    movel(p[x_c + -0.041312, y_c + 0.071568, z_c, rx, ry, rz], a, v)
    movel(p[x_c + -0.041015, y_c + 0.071951, z_c, rx, ry, rz], a, v)
    movel(p[x_c + -0.040710, y_c + 0.072343, z_c, rx, ry, rz], a, v)
    movel(p[x_c + -0.040396, y_c + 0.072744, z_c, rx, ry, rz], a, v)
    movel(p[x_c + -0.040073, y_c + 0.073156, z_c, rx, ry, rz], a, v)
    movel(p[x_c + -0.040073, y_c + 0.073156, z_c, rx, ry, rz], a, v)
    movel(p[x_c + -0.039958, y_c + 0.073302, z_c, rx, ry, rz], a, v)
    movel(p[x_c + -0.039844, y_c + 0.073448, z_c, rx, ry, rz], a, v)
    movel(p[x_c + -0.039729, y_c + 0.073594, z_c, rx, ry, rz], a, v)
    movel(p[x_c + -0.039615, y_c + 0.073740, z_c, rx, ry, rz], a, v)
    movel(p[x_c + -0.039501, y_c + 0.073885, z_c, rx, ry, rz], a, v)
    movel(p[x_c + -0.039388, y_c + 0.074029, z_c, rx, ry, rz], a, v)
    movel(p[x_c + -0.039276, y_c + 0.074172, z_c, rx, ry, rz], a, v)
    movel(p[x_c + -0.039164, y_c + 0.074315, z_c, rx, ry, rz], a, v)
    movel(p[x_c + -0.039053, y_c + 0.074457, z_c, rx, ry, rz], a, v)
    movel(p[x_c + -0.038942, y_c + 0.074597, z_c, rx, ry, rz], a, v)
    movel(p[x_c + -0.038833, y_c + 0.074737, z_c, rx, ry, rz], a, v)
    movel(p[x_c + -0.038724, y_c + 0.074876, z_c, rx, ry, rz], a, v)
    movel(p[x_c + -0.038617, y_c + 0.075013, z_c, rx, ry, rz], a, v)
    movel(p[x_c + -0.038511, y_c + 0.075148, z_c, rx, ry, rz], a, v)
    movel(p[x_c + -0.038405, y_c + 0.075283, z_c, rx, ry, rz], a, v)
    movel(p[x_c + -0.038301, y_c + 0.075416, z_c, rx, ry, rz], a, v)
    movel(p[x_c + -0.038199, y_c + 0.075547, z_c, rx, ry, rz], a, v)
    movel(p[x_c + -0.038098, y_c + 0.075676, z_c, rx, ry, rz], a, v)
    movel(p[x_c + -0.037998, y_c + 0.075804, z_c, rx, ry, rz], a, v)
    movel(p[x_c + -0.037900, y_c + 0.075929, z_c, rx, ry, rz], a, v)
    movel(p[x_c + -0.037803, y_c + 0.076053, z_c, rx, ry, rz], a, v)
    movel(p[x_c + -0.037708, y_c + 0.076174, z_c, rx, ry, rz], a, v)
    movel(p[x_c + -0.037615, y_c + 0.076294, z_c, rx, ry, rz], a, v)
    movel(p[x_c + -0.037523, y_c + 0.076411, z_c, rx, ry, rz], a, v)
    movel(p[x_c + -0.037434, y_c + 0.076525, z_c, rx, ry, rz], a, v)
    movel(p[x_c + -0.037346, y_c + 0.076637, z_c, rx, ry, rz], a, v)
    movel(p[x_c + -0.037261, y_c + 0.076747, z_c, rx, ry, rz], a, v)
    movel(p[x_c + -0.037177, y_c + 0.076854, z_c, rx, ry, rz], a, v)
    movel(p[x_c + -0.037096, y_c + 0.076958, z_c, rx, ry, rz], a, v)
    movel(p[x_c + -0.037017, y_c + 0.077059, z_c, rx, ry, rz], a, v)
    movel(p[x_c + -0.036940, y_c + 0.077157, z_c, rx, ry, rz], a, v)
    movel(p[x_c + -0.036866, y_c + 0.077253, z_c, rx, ry, rz], a, v)
    movel(p[x_c + -0.036794, y_c + 0.077345, z_c, rx, ry, rz], a, v)
    movel(p[x_c + -0.036725, y_c + 0.077434, z_c, rx, ry, rz], a, v)
    movel(p[x_c + -0.036658, y_c + 0.077519, z_c, rx, ry, rz], a, v)
    movel(p[x_c + -0.036594, y_c + 0.077602, z_c, rx, ry, rz], a, v)
    movel(p[x_c + -0.036533, y_c + 0.077680, z_c, rx, ry, rz], a, v)
    movel(p[x_c + -0.036475, y_c + 0.077755, z_c, rx, ry, rz], a, v)
    movel(p[x_c + -0.036419, y_c + 0.077827, z_c, rx, ry, rz], a, v)
    movel(p[x_c + -0.036367, y_c + 0.077895, z_c, rx, ry, rz], a, v)
    movel(p[x_c + -0.036317, y_c + 0.077959, z_c, rx, ry, rz], a, v)
    movel(p[x_c + -0.036271, y_c + 0.078018, z_c, rx, ry, rz], a, v)
    movel(p[x_c + -0.036227, y_c + 0.078074, z_c, rx, ry, rz], a, v)
    movel(p[x_c + -0.036188, y_c + 0.078126, z_c, rx, ry, rz], a, v)
    movel(p[x_c + -0.036151, y_c + 0.078173, z_c, rx, ry, rz], a, v)
    movel(p[x_c + -0.036118, y_c + 0.078217, z_c, rx, ry, rz], a, v)
    movel(p[x_c + -0.036088, y_c + 0.078255, z_c, rx, ry, rz], a, v)
    movel(p[x_c + -0.036062, y_c + 0.078290, z_c, rx, ry, rz], a, v)
    movel(p[x_c + -0.036039, y_c + 0.078319, z_c, rx, ry, rz], a, v)
    movel(p[x_c + -0.036039, y_c + 0.078319, z_c, rx, ry, rz], a, v)
    movel(p[x_c + -0.035423, y_c + 0.079129, z_c, rx, ry, rz], a, v)
    movel(p[x_c + -0.035423, y_c + 0.079129, z_c, rx, ry, rz], a, v)
    movel(p[x_c + -0.037378, y_c + 0.080396, z_c, rx, ry, rz], a, v)
    movel(p[x_c + -0.037378, y_c + 0.080396, z_c, rx, ry, rz], a, v)
    movel(p[x_c + -0.037680, y_c + 0.080589, z_c, rx, ry, rz], a, v)
    movel(p[x_c + -0.037987, y_c + 0.080780, z_c, rx, ry, rz], a, v)
    movel(p[x_c + -0.038299, y_c + 0.080970, z_c, rx, ry, rz], a, v)
    movel(p[x_c + -0.038617, y_c + 0.081159, z_c, rx, ry, rz], a, v)
    movel(p[x_c + -0.038940, y_c + 0.081346, z_c, rx, ry, rz], a, v)
    movel(p[x_c + -0.039269, y_c + 0.081532, z_c, rx, ry, rz], a, v)
    movel(p[x_c + -0.039602, y_c + 0.081716, z_c, rx, ry, rz], a, v)
    movel(p[x_c + -0.039939, y_c + 0.081898, z_c, rx, ry, rz], a, v)
    movel(p[x_c + -0.040281, y_c + 0.082078, z_c, rx, ry, rz], a, v)
    movel(p[x_c + -0.040628, y_c + 0.082257, z_c, rx, ry, rz], a, v)
    movel(p[x_c + -0.040978, y_c + 0.082434, z_c, rx, ry, rz], a, v)
    movel(p[x_c + -0.041332, y_c + 0.082609, z_c, rx, ry, rz], a, v)
    movel(p[x_c + -0.041690, y_c + 0.082782, z_c, rx, ry, rz], a, v)
    movel(p[x_c + -0.042052, y_c + 0.082952, z_c, rx, ry, rz], a, v)
    movel(p[x_c + -0.042417, y_c + 0.083121, z_c, rx, ry, rz], a, v)
    movel(p[x_c + -0.042785, y_c + 0.083287, z_c, rx, ry, rz], a, v)
    movel(p[x_c + -0.043157, y_c + 0.083452, z_c, rx, ry, rz], a, v)
    movel(p[x_c + -0.043531, y_c + 0.083613, z_c, rx, ry, rz], a, v)
    movel(p[x_c + -0.043908, y_c + 0.083773, z_c, rx, ry, rz], a, v)
    movel(p[x_c + -0.044287, y_c + 0.083930, z_c, rx, ry, rz], a, v)
    movel(p[x_c + -0.044668, y_c + 0.084084, z_c, rx, ry, rz], a, v)
    movel(p[x_c + -0.045052, y_c + 0.084236, z_c, rx, ry, rz], a, v)
    movel(p[x_c + -0.045438, y_c + 0.084385, z_c, rx, ry, rz], a, v)
    movel(p[x_c + -0.045825, y_c + 0.084531, z_c, rx, ry, rz], a, v)
    movel(p[x_c + -0.046214, y_c + 0.084674, z_c, rx, ry, rz], a, v)
    movel(p[x_c + -0.046604, y_c + 0.084815, z_c, rx, ry, rz], a, v)
    movel(p[x_c + -0.046996, y_c + 0.084952, z_c, rx, ry, rz], a, v)
    movel(p[x_c + -0.047388, y_c + 0.085087, z_c, rx, ry, rz], a, v)
    movel(p[x_c + -0.047782, y_c + 0.085219, z_c, rx, ry, rz], a, v)
    movel(p[x_c + -0.048176, y_c + 0.085347, z_c, rx, ry, rz], a, v)
    movel(p[x_c + -0.048571, y_c + 0.085472, z_c, rx, ry, rz], a, v)
    movel(p[x_c + -0.048966, y_c + 0.085594, z_c, rx, ry, rz], a, v)
    movel(p[x_c + -0.049361, y_c + 0.085713, z_c, rx, ry, rz], a, v)
    movel(p[x_c + -0.049756, y_c + 0.085828, z_c, rx, ry, rz], a, v)
    movel(p[x_c + -0.050151, y_c + 0.085939, z_c, rx, ry, rz], a, v)
    movel(p[x_c + -0.050545, y_c + 0.086047, z_c, rx, ry, rz], a, v)
    movel(p[x_c + -0.050939, y_c + 0.086152, z_c, rx, ry, rz], a, v)
    movel(p[x_c + -0.051332, y_c + 0.086253, z_c, rx, ry, rz], a, v)
    movel(p[x_c + -0.051724, y_c + 0.086350, z_c, rx, ry, rz], a, v)
    movel(p[x_c + -0.052115, y_c + 0.086443, z_c, rx, ry, rz], a, v)
    movel(p[x_c + -0.052505, y_c + 0.086532, z_c, rx, ry, rz], a, v)
    movel(p[x_c + -0.052893, y_c + 0.086618, z_c, rx, ry, rz], a, v)
    movel(p[x_c + -0.053280, y_c + 0.086699, z_c, rx, ry, rz], a, v)
    movel(p[x_c + -0.053665, y_c + 0.086777, z_c, rx, ry, rz], a, v)
    movel(p[x_c + -0.054047, y_c + 0.086850, z_c, rx, ry, rz], a, v)
    movel(p[x_c + -0.054428, y_c + 0.086919, z_c, rx, ry, rz], a, v)
    movel(p[x_c + -0.054806, y_c + 0.086984, z_c, rx, ry, rz], a, v)
    movel(p[x_c + -0.055182, y_c + 0.087044, z_c, rx, ry, rz], a, v)
    movel(p[x_c + -0.055554, y_c + 0.087100, z_c, rx, ry, rz], a, v)
    movel(p[x_c + -0.055554, y_c + 0.087100, z_c, rx, ry, rz], a, v)
    movel(p[x_c + -0.055822, y_c + 0.087137, z_c, rx, ry, rz], a, v)
    movel(p[x_c + -0.056094, y_c + 0.087172, z_c, rx, ry, rz], a, v)
    movel(p[x_c + -0.056371, y_c + 0.087205, z_c, rx, ry, rz], a, v)
    movel(p[x_c + -0.056652, y_c + 0.087236, z_c, rx, ry, rz], a, v)
    movel(p[x_c + -0.056937, y_c + 0.087265, z_c, rx, ry, rz], a, v)
    movel(p[x_c + -0.057226, y_c + 0.087292, z_c, rx, ry, rz], a, v)
    movel(p[x_c + -0.057519, y_c + 0.087317, z_c, rx, ry, rz], a, v)
    movel(p[x_c + -0.057816, y_c + 0.087340, z_c, rx, ry, rz], a, v)
    movel(p[x_c + -0.058116, y_c + 0.087360, z_c, rx, ry, rz], a, v)
    movel(p[x_c + -0.058421, y_c + 0.087379, z_c, rx, ry, rz], a, v)
    movel(p[x_c + -0.058728, y_c + 0.087395, z_c, rx, ry, rz], a, v)
    movel(p[x_c + -0.059039, y_c + 0.087410, z_c, rx, ry, rz], a, v)
    movel(p[x_c + -0.059354, y_c + 0.087422, z_c, rx, ry, rz], a, v)
    movel(p[x_c + -0.059671, y_c + 0.087432, z_c, rx, ry, rz], a, v)
    movel(p[x_c + -0.059991, y_c + 0.087441, z_c, rx, ry, rz], a, v)
    movel(p[x_c + -0.060315, y_c + 0.087447, z_c, rx, ry, rz], a, v)
    movel(p[x_c + -0.060641, y_c + 0.087451, z_c, rx, ry, rz], a, v)
    movel(p[x_c + -0.060969, y_c + 0.087453, z_c, rx, ry, rz], a, v)
    movel(p[x_c + -0.061300, y_c + 0.087453, z_c, rx, ry, rz], a, v)
    movel(p[x_c + -0.061634, y_c + 0.087451, z_c, rx, ry, rz], a, v)
    movel(p[x_c + -0.061970, y_c + 0.087447, z_c, rx, ry, rz], a, v)
    movel(p[x_c + -0.062308, y_c + 0.087441, z_c, rx, ry, rz], a, v)
    movel(p[x_c + -0.062648, y_c + 0.087433, z_c, rx, ry, rz], a, v)
    movel(p[x_c + -0.062990, y_c + 0.087423, z_c, rx, ry, rz], a, v)
    movel(p[x_c + -0.063334, y_c + 0.087411, z_c, rx, ry, rz], a, v)
    movel(p[x_c + -0.063679, y_c + 0.087397, z_c, rx, ry, rz], a, v)
    movel(p[x_c + -0.064027, y_c + 0.087381, z_c, rx, ry, rz], a, v)
    movel(p[x_c + -0.064375, y_c + 0.087363, z_c, rx, ry, rz], a, v)
    movel(p[x_c + -0.064725, y_c + 0.087343, z_c, rx, ry, rz], a, v)
    movel(p[x_c + -0.065076, y_c + 0.087321, z_c, rx, ry, rz], a, v)
    movel(p[x_c + -0.065428, y_c + 0.087297, z_c, rx, ry, rz], a, v)
    movel(p[x_c + -0.065782, y_c + 0.087271, z_c, rx, ry, rz], a, v)
    movel(p[x_c + -0.066136, y_c + 0.087243, z_c, rx, ry, rz], a, v)
    movel(p[x_c + -0.066491, y_c + 0.087213, z_c, rx, ry, rz], a, v)
    movel(p[x_c + -0.066846, y_c + 0.087181, z_c, rx, ry, rz], a, v)
    movel(p[x_c + -0.067202, y_c + 0.087148, z_c, rx, ry, rz], a, v)
    movel(p[x_c + -0.067558, y_c + 0.087112, z_c, rx, ry, rz], a, v)
    movel(p[x_c + -0.067915, y_c + 0.087074, z_c, rx, ry, rz], a, v)
    movel(p[x_c + -0.068272, y_c + 0.087034, z_c, rx, ry, rz], a, v)
    movel(p[x_c + -0.068629, y_c + 0.086993, z_c, rx, ry, rz], a, v)
    movel(p[x_c + -0.068985, y_c + 0.086949, z_c, rx, ry, rz], a, v)
    movel(p[x_c + -0.069342, y_c + 0.086904, z_c, rx, ry, rz], a, v)
    movel(p[x_c + -0.069698, y_c + 0.086856, z_c, rx, ry, rz], a, v)
    movel(p[x_c + -0.070054, y_c + 0.086807, z_c, rx, ry, rz], a, v)
    movel(p[x_c + -0.070409, y_c + 0.086755, z_c, rx, ry, rz], a, v)
    movel(p[x_c + -0.070764, y_c + 0.086702, z_c, rx, ry, rz], a, v)
    movel(p[x_c + -0.071117, y_c + 0.086647, z_c, rx, ry, rz], a, v)
    movel(p[x_c + -0.071470, y_c + 0.086590, z_c, rx, ry, rz], a, v)
    movel(p[x_c + -0.071822, y_c + 0.086531, z_c, rx, ry, rz], a, v)
    movel(p[x_c + -0.071822, y_c + 0.086531, z_c, rx, ry, rz], a, v)
    movel(p[x_c + -0.071990, y_c + 0.086502, z_c, rx, ry, rz], a, v)
    movel(p[x_c + -0.072167, y_c + 0.086470, z_c, rx, ry, rz], a, v)
    movel(p[x_c + -0.072353, y_c + 0.086437, z_c, rx, ry, rz], a, v)
    movel(p[x_c + -0.072546, y_c + 0.086401, z_c, rx, ry, rz], a, v)
    movel(p[x_c + -0.072747, y_c + 0.086363, z_c, rx, ry, rz], a, v)
    movel(p[x_c + -0.072956, y_c + 0.086323, z_c, rx, ry, rz], a, v)
    movel(p[x_c + -0.073172, y_c + 0.086281, z_c, rx, ry, rz], a, v)
    movel(p[x_c + -0.073394, y_c + 0.086237, z_c, rx, ry, rz], a, v)
    movel(p[x_c + -0.073623, y_c + 0.086191, z_c, rx, ry, rz], a, v)
    movel(p[x_c + -0.073857, y_c + 0.086144, z_c, rx, ry, rz], a, v)
    movel(p[x_c + -0.074097, y_c + 0.086095, z_c, rx, ry, rz], a, v)
    movel(p[x_c + -0.074342, y_c + 0.086045, z_c, rx, ry, rz], a, v)
    movel(p[x_c + -0.074591, y_c + 0.085993, z_c, rx, ry, rz], a, v)
    movel(p[x_c + -0.074845, y_c + 0.085940, z_c, rx, ry, rz], a, v)
    movel(p[x_c + -0.075103, y_c + 0.085885, z_c, rx, ry, rz], a, v)
    movel(p[x_c + -0.075365, y_c + 0.085830, z_c, rx, ry, rz], a, v)
    movel(p[x_c + -0.075629, y_c + 0.085773, z_c, rx, ry, rz], a, v)
    movel(p[x_c + -0.075897, y_c + 0.085716, z_c, rx, ry, rz], a, v)
    movel(p[x_c + -0.076166, y_c + 0.085657, z_c, rx, ry, rz], a, v)
    movel(p[x_c + -0.076438, y_c + 0.085598, z_c, rx, ry, rz], a, v)
    movel(p[x_c + -0.076712, y_c + 0.085538, z_c, rx, ry, rz], a, v)
    movel(p[x_c + -0.076986, y_c + 0.085477, z_c, rx, ry, rz], a, v)
    movel(p[x_c + -0.077262, y_c + 0.085416, z_c, rx, ry, rz], a, v)
    movel(p[x_c + -0.077538, y_c + 0.085354, z_c, rx, ry, rz], a, v)
    movel(p[x_c + -0.077814, y_c + 0.085292, z_c, rx, ry, rz], a, v)
    movel(p[x_c + -0.078090, y_c + 0.085229, z_c, rx, ry, rz], a, v)
    movel(p[x_c + -0.078365, y_c + 0.085167, z_c, rx, ry, rz], a, v)
    movel(p[x_c + -0.078640, y_c + 0.085104, z_c, rx, ry, rz], a, v)
    movel(p[x_c + -0.078912, y_c + 0.085041, z_c, rx, ry, rz], a, v)
    movel(p[x_c + -0.079184, y_c + 0.084978, z_c, rx, ry, rz], a, v)
    movel(p[x_c + -0.079452, y_c + 0.084916, z_c, rx, ry, rz], a, v)
    movel(p[x_c + -0.079719, y_c + 0.084853, z_c, rx, ry, rz], a, v)
    movel(p[x_c + -0.079982, y_c + 0.084791, z_c, rx, ry, rz], a, v)
    movel(p[x_c + -0.080242, y_c + 0.084729, z_c, rx, ry, rz], a, v)
    movel(p[x_c + -0.080499, y_c + 0.084668, z_c, rx, ry, rz], a, v)
    movel(p[x_c + -0.080751, y_c + 0.084607, z_c, rx, ry, rz], a, v)
    movel(p[x_c + -0.080999, y_c + 0.084547, z_c, rx, ry, rz], a, v)
    movel(p[x_c + -0.081242, y_c + 0.084488, z_c, rx, ry, rz], a, v)
    movel(p[x_c + -0.081480, y_c + 0.084429, z_c, rx, ry, rz], a, v)
    movel(p[x_c + -0.081712, y_c + 0.084372, z_c, rx, ry, rz], a, v)
    movel(p[x_c + -0.081938, y_c + 0.084315, z_c, rx, ry, rz], a, v)
    movel(p[x_c + -0.082158, y_c + 0.084259, z_c, rx, ry, rz], a, v)
    movel(p[x_c + -0.082371, y_c + 0.084205, z_c, rx, ry, rz], a, v)
    movel(p[x_c + -0.082577, y_c + 0.084152, z_c, rx, ry, rz], a, v)
    movel(p[x_c + -0.082775, y_c + 0.084100, z_c, rx, ry, rz], a, v)
    movel(p[x_c + -0.082965, y_c + 0.084049, z_c, rx, ry, rz], a, v)
    movel(p[x_c + -0.083148, y_c + 0.084000, z_c, rx, ry, rz], a, v)
    movel(p[x_c + -0.083321, y_c + 0.083953, z_c, rx, ry, rz], a, v)
    movel(p[x_c + -0.083486, y_c + 0.083907, z_c, rx, ry, rz], a, v)
    movel(p[x_c + -0.083486, y_c + 0.083907, z_c, rx, ry, rz], a, v)
    movel(p[x_c + -0.083592, y_c + 0.083878, z_c, rx, ry, rz], a, v)
    movel(p[x_c + -0.083694, y_c + 0.083849, z_c, rx, ry, rz], a, v)
    movel(p[x_c + -0.083792, y_c + 0.083822, z_c, rx, ry, rz], a, v)
    movel(p[x_c + -0.083885, y_c + 0.083797, z_c, rx, ry, rz], a, v)
    movel(p[x_c + -0.083974, y_c + 0.083773, z_c, rx, ry, rz], a, v)
    movel(p[x_c + -0.084059, y_c + 0.083750, z_c, rx, ry, rz], a, v)
    movel(p[x_c + -0.084140, y_c + 0.083730, z_c, rx, ry, rz], a, v)
    movel(p[x_c + -0.084217, y_c + 0.083711, z_c, rx, ry, rz], a, v)
    movel(p[x_c + -0.084290, y_c + 0.083695, z_c, rx, ry, rz], a, v)
    movel(p[x_c + -0.084359, y_c + 0.083680, z_c, rx, ry, rz], a, v)
    movel(p[x_c + -0.084424, y_c + 0.083667, z_c, rx, ry, rz], a, v)
    movel(p[x_c + -0.084485, y_c + 0.083657, z_c, rx, ry, rz], a, v)
    movel(p[x_c + -0.084543, y_c + 0.083649, z_c, rx, ry, rz], a, v)
    movel(p[x_c + -0.084597, y_c + 0.083643, z_c, rx, ry, rz], a, v)
    movel(p[x_c + -0.084647, y_c + 0.083640, z_c, rx, ry, rz], a, v)
    movel(p[x_c + -0.084693, y_c + 0.083639, z_c, rx, ry, rz], a, v)
    movel(p[x_c + -0.084736, y_c + 0.083641, z_c, rx, ry, rz], a, v)
    movel(p[x_c + -0.084776, y_c + 0.083646, z_c, rx, ry, rz], a, v)
    movel(p[x_c + -0.084812, y_c + 0.083654, z_c, rx, ry, rz], a, v)
    movel(p[x_c + -0.084845, y_c + 0.083664, z_c, rx, ry, rz], a, v)
    movel(p[x_c + -0.084875, y_c + 0.083677, z_c, rx, ry, rz], a, v)
    movel(p[x_c + -0.084901, y_c + 0.083694, z_c, rx, ry, rz], a, v)
    movel(p[x_c + -0.084924, y_c + 0.083713, z_c, rx, ry, rz], a, v)
    movel(p[x_c + -0.084944, y_c + 0.083736, z_c, rx, ry, rz], a, v)
    movel(p[x_c + -0.084961, y_c + 0.083762, z_c, rx, ry, rz], a, v)
    movel(p[x_c + -0.084974, y_c + 0.083791, z_c, rx, ry, rz], a, v)
    movel(p[x_c + -0.084985, y_c + 0.083824, z_c, rx, ry, rz], a, v)
    movel(p[x_c + -0.084993, y_c + 0.083861, z_c, rx, ry, rz], a, v)
    movel(p[x_c + -0.084998, y_c + 0.083901, z_c, rx, ry, rz], a, v)
    movel(p[x_c + -0.085000, y_c + 0.083945, z_c, rx, ry, rz], a, v)
    movel(p[x_c + -0.084999, y_c + 0.083993, z_c, rx, ry, rz], a, v)
    movel(p[x_c + -0.084996, y_c + 0.084044, z_c, rx, ry, rz], a, v)
    movel(p[x_c + -0.084990, y_c + 0.084100, z_c, rx, ry, rz], a, v)
    movel(p[x_c + -0.084982, y_c + 0.084160, z_c, rx, ry, rz], a, v)
    movel(p[x_c + -0.084971, y_c + 0.084224, z_c, rx, ry, rz], a, v)
    movel(p[x_c + -0.084957, y_c + 0.084292, z_c, rx, ry, rz], a, v)
    movel(p[x_c + -0.084941, y_c + 0.084364, z_c, rx, ry, rz], a, v)
    movel(p[x_c + -0.084923, y_c + 0.084441, z_c, rx, ry, rz], a, v)
    movel(p[x_c + -0.084902, y_c + 0.084523, z_c, rx, ry, rz], a, v)
    movel(p[x_c + -0.084879, y_c + 0.084609, z_c, rx, ry, rz], a, v)
    movel(p[x_c + -0.084854, y_c + 0.084700, z_c, rx, ry, rz], a, v)
    movel(p[x_c + -0.084827, y_c + 0.084795, z_c, rx, ry, rz], a, v)
    movel(p[x_c + -0.084797, y_c + 0.084895, z_c, rx, ry, rz], a, v)
    movel(p[x_c + -0.084766, y_c + 0.085001, z_c, rx, ry, rz], a, v)
    movel(p[x_c + -0.084732, y_c + 0.085111, z_c, rx, ry, rz], a, v)
    movel(p[x_c + -0.084697, y_c + 0.085227, z_c, rx, ry, rz], a, v)
    movel(p[x_c + -0.084660, y_c + 0.085347, z_c, rx, ry, rz], a, v)
    movel(p[x_c + -0.084621, y_c + 0.085473, z_c, rx, ry, rz], a, v)
    movel(p[x_c + -0.084580, y_c + 0.085605, z_c, rx, ry, rz], a, v)
    movel(p[x_c + -0.084580, y_c + 0.085605, z_c, rx, ry, rz], a, v)
    movel(p[x_c + -0.084501, y_c + 0.085849, z_c, rx, ry, rz], a, v)
    movel(p[x_c + -0.084416, y_c + 0.086090, z_c, rx, ry, rz], a, v)
    movel(p[x_c + -0.084326, y_c + 0.086328, z_c, rx, ry, rz], a, v)
    movel(p[x_c + -0.084230, y_c + 0.086563, z_c, rx, ry, rz], a, v)
    movel(p[x_c + -0.084128, y_c + 0.086796, z_c, rx, ry, rz], a, v)
    movel(p[x_c + -0.084020, y_c + 0.087025, z_c, rx, ry, rz], a, v)
    movel(p[x_c + -0.083907, y_c + 0.087252, z_c, rx, ry, rz], a, v)
    movel(p[x_c + -0.083787, y_c + 0.087477, z_c, rx, ry, rz], a, v)
    movel(p[x_c + -0.083661, y_c + 0.087699, z_c, rx, ry, rz], a, v)
    movel(p[x_c + -0.083528, y_c + 0.087919, z_c, rx, ry, rz], a, v)
    movel(p[x_c + -0.083389, y_c + 0.088137, z_c, rx, ry, rz], a, v)
    movel(p[x_c + -0.083243, y_c + 0.088353, z_c, rx, ry, rz], a, v)
    movel(p[x_c + -0.083090, y_c + 0.088567, z_c, rx, ry, rz], a, v)
    movel(p[x_c + -0.082931, y_c + 0.088778, z_c, rx, ry, rz], a, v)
    movel(p[x_c + -0.082764, y_c + 0.088988, z_c, rx, ry, rz], a, v)
    movel(p[x_c + -0.082591, y_c + 0.089197, z_c, rx, ry, rz], a, v)
    movel(p[x_c + -0.082410, y_c + 0.089403, z_c, rx, ry, rz], a, v)
    movel(p[x_c + -0.082221, y_c + 0.089609, z_c, rx, ry, rz], a, v)
    movel(p[x_c + -0.082025, y_c + 0.089812, z_c, rx, ry, rz], a, v)
    movel(p[x_c + -0.081822, y_c + 0.090015, z_c, rx, ry, rz], a, v)
    movel(p[x_c + -0.081611, y_c + 0.090216, z_c, rx, ry, rz], a, v)
    movel(p[x_c + -0.081391, y_c + 0.090416, z_c, rx, ry, rz], a, v)
    movel(p[x_c + -0.081164, y_c + 0.090616, z_c, rx, ry, rz], a, v)
    movel(p[x_c + -0.080929, y_c + 0.090814, z_c, rx, ry, rz], a, v)
    movel(p[x_c + -0.080685, y_c + 0.091011, z_c, rx, ry, rz], a, v)
    movel(p[x_c + -0.080433, y_c + 0.091208, z_c, rx, ry, rz], a, v)
    movel(p[x_c + -0.080173, y_c + 0.091404, z_c, rx, ry, rz], a, v)
    movel(p[x_c + -0.079904, y_c + 0.091600, z_c, rx, ry, rz], a, v)
    movel(p[x_c + -0.079626, y_c + 0.091795, z_c, rx, ry, rz], a, v)
    movel(p[x_c + -0.079339, y_c + 0.091990, z_c, rx, ry, rz], a, v)
    movel(p[x_c + -0.079044, y_c + 0.092185, z_c, rx, ry, rz], a, v)
    movel(p[x_c + -0.078739, y_c + 0.092379, z_c, rx, ry, rz], a, v)
    movel(p[x_c + -0.078425, y_c + 0.092574, z_c, rx, ry, rz], a, v)
    movel(p[x_c + -0.078102, y_c + 0.092768, z_c, rx, ry, rz], a, v)
    movel(p[x_c + -0.077769, y_c + 0.092963, z_c, rx, ry, rz], a, v)
    movel(p[x_c + -0.077427, y_c + 0.093158, z_c, rx, ry, rz], a, v)
    movel(p[x_c + -0.077074, y_c + 0.093353, z_c, rx, ry, rz], a, v)
    movel(p[x_c + -0.076713, y_c + 0.093549, z_c, rx, ry, rz], a, v)
    movel(p[x_c + -0.076341, y_c + 0.093746, z_c, rx, ry, rz], a, v)
    movel(p[x_c + -0.075959, y_c + 0.093943, z_c, rx, ry, rz], a, v)
    movel(p[x_c + -0.075567, y_c + 0.094141, z_c, rx, ry, rz], a, v)
    movel(p[x_c + -0.075164, y_c + 0.094340, z_c, rx, ry, rz], a, v)
    movel(p[x_c + -0.074751, y_c + 0.094539, z_c, rx, ry, rz], a, v)
    movel(p[x_c + -0.074328, y_c + 0.094740, z_c, rx, ry, rz], a, v)
    movel(p[x_c + -0.073893, y_c + 0.094942, z_c, rx, ry, rz], a, v)
    movel(p[x_c + -0.073448, y_c + 0.095145, z_c, rx, ry, rz], a, v)
    movel(p[x_c + -0.072993, y_c + 0.095350, z_c, rx, ry, rz], a, v)
    movel(p[x_c + -0.072526, y_c + 0.095556, z_c, rx, ry, rz], a, v)
    movel(p[x_c + -0.072047, y_c + 0.095763, z_c, rx, ry, rz], a, v)
    movel(p[x_c + -0.072047, y_c + 0.095763, z_c, rx, ry, rz], a, v)
    movel(p[x_c + -0.071476, y_c + 0.096010, z_c, rx, ry, rz], a, v)
    movel(p[x_c + -0.070926, y_c + 0.096248, z_c, rx, ry, rz], a, v)
    movel(p[x_c + -0.070396, y_c + 0.096478, z_c, rx, ry, rz], a, v)
    movel(p[x_c + -0.069886, y_c + 0.096700, z_c, rx, ry, rz], a, v)
    movel(p[x_c + -0.069395, y_c + 0.096916, z_c, rx, ry, rz], a, v)
    movel(p[x_c + -0.068921, y_c + 0.097125, z_c, rx, ry, rz], a, v)
    movel(p[x_c + -0.068465, y_c + 0.097329, z_c, rx, ry, rz], a, v)
    movel(p[x_c + -0.068026, y_c + 0.097527, z_c, rx, ry, rz], a, v)
    movel(p[x_c + -0.067602, y_c + 0.097721, z_c, rx, ry, rz], a, v)
    movel(p[x_c + -0.067193, y_c + 0.097911, z_c, rx, ry, rz], a, v)
    movel(p[x_c + -0.066798, y_c + 0.098097, z_c, rx, ry, rz], a, v)
    movel(p[x_c + -0.066416, y_c + 0.098280, z_c, rx, ry, rz], a, v)
    movel(p[x_c + -0.066046, y_c + 0.098460, z_c, rx, ry, rz], a, v)
    movel(p[x_c + -0.065688, y_c + 0.098639, z_c, rx, ry, rz], a, v)
    movel(p[x_c + -0.065342, y_c + 0.098816, z_c, rx, ry, rz], a, v)
    movel(p[x_c + -0.065005, y_c + 0.098992, z_c, rx, ry, rz], a, v)
    movel(p[x_c + -0.064677, y_c + 0.099168, z_c, rx, ry, rz], a, v)
    movel(p[x_c + -0.064358, y_c + 0.099344, z_c, rx, ry, rz], a, v)
    movel(p[x_c + -0.064046, y_c + 0.099521, z_c, rx, ry, rz], a, v)
    movel(p[x_c + -0.063742, y_c + 0.099699, z_c, rx, ry, rz], a, v)
    movel(p[x_c + -0.063443, y_c + 0.099879, z_c, rx, ry, rz], a, v)
    movel(p[x_c + -0.063150, y_c + 0.100062, z_c, rx, ry, rz], a, v)
    movel(p[x_c + -0.062861, y_c + 0.100247, z_c, rx, ry, rz], a, v)
    movel(p[x_c + -0.062576, y_c + 0.100436, z_c, rx, ry, rz], a, v)
    movel(p[x_c + -0.062293, y_c + 0.100629, z_c, rx, ry, rz], a, v)
    movel(p[x_c + -0.062013, y_c + 0.100827, z_c, rx, ry, rz], a, v)
    movel(p[x_c + -0.061734, y_c + 0.101029, z_c, rx, ry, rz], a, v)
    movel(p[x_c + -0.061456, y_c + 0.101238, z_c, rx, ry, rz], a, v)
    movel(p[x_c + -0.061177, y_c + 0.101453, z_c, rx, ry, rz], a, v)
    movel(p[x_c + -0.060897, y_c + 0.101674, z_c, rx, ry, rz], a, v)
    movel(p[x_c + -0.060615, y_c + 0.101903, z_c, rx, ry, rz], a, v)
    movel(p[x_c + -0.060330, y_c + 0.102139, z_c, rx, ry, rz], a, v)
    movel(p[x_c + -0.060042, y_c + 0.102384, z_c, rx, ry, rz], a, v)
    movel(p[x_c + -0.059750, y_c + 0.102638, z_c, rx, ry, rz], a, v)
    movel(p[x_c + -0.059453, y_c + 0.102902, z_c, rx, ry, rz], a, v)
    movel(p[x_c + -0.059149, y_c + 0.103175, z_c, rx, ry, rz], a, v)
    movel(p[x_c + -0.058839, y_c + 0.103459, z_c, rx, ry, rz], a, v)
    movel(p[x_c + -0.058521, y_c + 0.103754, z_c, rx, ry, rz], a, v)
    movel(p[x_c + -0.058196, y_c + 0.104061, z_c, rx, ry, rz], a, v)
    movel(p[x_c + -0.057861, y_c + 0.104380, z_c, rx, ry, rz], a, v)
    movel(p[x_c + -0.057516, y_c + 0.104712, z_c, rx, ry, rz], a, v)
    movel(p[x_c + -0.057160, y_c + 0.105058, z_c, rx, ry, rz], a, v)
    movel(p[x_c + -0.056793, y_c + 0.105417, z_c, rx, ry, rz], a, v)
    movel(p[x_c + -0.056414, y_c + 0.105790, z_c, rx, ry, rz], a, v)
    movel(p[x_c + -0.056022, y_c + 0.106179, z_c, rx, ry, rz], a, v)
    movel(p[x_c + -0.055615, y_c + 0.106582, z_c, rx, ry, rz], a, v)
    movel(p[x_c + -0.055194, y_c + 0.107002, z_c, rx, ry, rz], a, v)
    movel(p[x_c + -0.054758, y_c + 0.107439, z_c, rx, ry, rz], a, v)
    movel(p[x_c + -0.054305, y_c + 0.107893, z_c, rx, ry, rz], a, v)
    movel(p[x_c + -0.054305, y_c + 0.107893, z_c, rx, ry, rz], a, v)
    movel(p[x_c + -0.054117, y_c + 0.108082, z_c, rx, ry, rz], a, v)
    movel(p[x_c + -0.053927, y_c + 0.108271, z_c, rx, ry, rz], a, v)
    movel(p[x_c + -0.053737, y_c + 0.108461, z_c, rx, ry, rz], a, v)
    movel(p[x_c + -0.053546, y_c + 0.108651, z_c, rx, ry, rz], a, v)
    movel(p[x_c + -0.053355, y_c + 0.108841, z_c, rx, ry, rz], a, v)
    movel(p[x_c + -0.053163, y_c + 0.109031, z_c, rx, ry, rz], a, v)
    movel(p[x_c + -0.052972, y_c + 0.109220, z_c, rx, ry, rz], a, v)
    movel(p[x_c + -0.052780, y_c + 0.109409, z_c, rx, ry, rz], a, v)
    movel(p[x_c + -0.052589, y_c + 0.109598, z_c, rx, ry, rz], a, v)
    movel(p[x_c + -0.052397, y_c + 0.109786, z_c, rx, ry, rz], a, v)
    movel(p[x_c + -0.052206, y_c + 0.109974, z_c, rx, ry, rz], a, v)
    movel(p[x_c + -0.052016, y_c + 0.110160, z_c, rx, ry, rz], a, v)
    movel(p[x_c + -0.051826, y_c + 0.110346, z_c, rx, ry, rz], a, v)
    movel(p[x_c + -0.051637, y_c + 0.110530, z_c, rx, ry, rz], a, v)
    movel(p[x_c + -0.051449, y_c + 0.110713, z_c, rx, ry, rz], a, v)
    movel(p[x_c + -0.051262, y_c + 0.110895, z_c, rx, ry, rz], a, v)
    movel(p[x_c + -0.051076, y_c + 0.111075, z_c, rx, ry, rz], a, v)
    movel(p[x_c + -0.050892, y_c + 0.111254, z_c, rx, ry, rz], a, v)
    movel(p[x_c + -0.050709, y_c + 0.111430, z_c, rx, ry, rz], a, v)
    movel(p[x_c + -0.050528, y_c + 0.111605, z_c, rx, ry, rz], a, v)
    movel(p[x_c + -0.050348, y_c + 0.111778, z_c, rx, ry, rz], a, v)
    movel(p[x_c + -0.050171, y_c + 0.111948, z_c, rx, ry, rz], a, v)
    movel(p[x_c + -0.049995, y_c + 0.112116, z_c, rx, ry, rz], a, v)
    movel(p[x_c + -0.049822, y_c + 0.112282, z_c, rx, ry, rz], a, v)
    movel(p[x_c + -0.049651, y_c + 0.112445, z_c, rx, ry, rz], a, v)
    movel(p[x_c + -0.049482, y_c + 0.112606, z_c, rx, ry, rz], a, v)
    movel(p[x_c + -0.049316, y_c + 0.112763, z_c, rx, ry, rz], a, v)
    movel(p[x_c + -0.049153, y_c + 0.112918, z_c, rx, ry, rz], a, v)
    movel(p[x_c + -0.048992, y_c + 0.113069, z_c, rx, ry, rz], a, v)
    movel(p[x_c + -0.048835, y_c + 0.113218, z_c, rx, ry, rz], a, v)
    movel(p[x_c + -0.048680, y_c + 0.113362, z_c, rx, ry, rz], a, v)
    movel(p[x_c + -0.048529, y_c + 0.113504, z_c, rx, ry, rz], a, v)
    movel(p[x_c + -0.048382, y_c + 0.113642, z_c, rx, ry, rz], a, v)
    movel(p[x_c + -0.048238, y_c + 0.113776, z_c, rx, ry, rz], a, v)
    movel(p[x_c + -0.048097, y_c + 0.113906, z_c, rx, ry, rz], a, v)
    movel(p[x_c + -0.047961, y_c + 0.114032, z_c, rx, ry, rz], a, v)
    movel(p[x_c + -0.047828, y_c + 0.114153, z_c, rx, ry, rz], a, v)
    movel(p[x_c + -0.047700, y_c + 0.114271, z_c, rx, ry, rz], a, v)
    movel(p[x_c + -0.047576, y_c + 0.114384, z_c, rx, ry, rz], a, v)
    movel(p[x_c + -0.047456, y_c + 0.114493, z_c, rx, ry, rz], a, v)
    movel(p[x_c + -0.047340, y_c + 0.114597, z_c, rx, ry, rz], a, v)
    movel(p[x_c + -0.047230, y_c + 0.114696, z_c, rx, ry, rz], a, v)
    movel(p[x_c + -0.047124, y_c + 0.114790, z_c, rx, ry, rz], a, v)
    movel(p[x_c + -0.047023, y_c + 0.114879, z_c, rx, ry, rz], a, v)
    movel(p[x_c + -0.046927, y_c + 0.114963, z_c, rx, ry, rz], a, v)
    movel(p[x_c + -0.046836, y_c + 0.115041, z_c, rx, ry, rz], a, v)
    movel(p[x_c + -0.046751, y_c + 0.115115, z_c, rx, ry, rz], a, v)
    movel(p[x_c + -0.046671, y_c + 0.115182, z_c, rx, ry, rz], a, v)
    movel(p[x_c + -0.046597, y_c + 0.115244, z_c, rx, ry, rz], a, v)
    movel(p[x_c + -0.046597, y_c + 0.115244, z_c, rx, ry, rz], a, v)
    movel(p[x_c + -0.046334, y_c + 0.115459, z_c, rx, ry, rz], a, v)
    movel(p[x_c + -0.046070, y_c + 0.115672, z_c, rx, ry, rz], a, v)
    movel(p[x_c + -0.045805, y_c + 0.115883, z_c, rx, ry, rz], a, v)
    movel(p[x_c + -0.045540, y_c + 0.116091, z_c, rx, ry, rz], a, v)
    movel(p[x_c + -0.045275, y_c + 0.116298, z_c, rx, ry, rz], a, v)
    movel(p[x_c + -0.045009, y_c + 0.116502, z_c, rx, ry, rz], a, v)
    movel(p[x_c + -0.044742, y_c + 0.116703, z_c, rx, ry, rz], a, v)
    movel(p[x_c + -0.044475, y_c + 0.116903, z_c, rx, ry, rz], a, v)
    movel(p[x_c + -0.044208, y_c + 0.117100, z_c, rx, ry, rz], a, v)
    movel(p[x_c + -0.043940, y_c + 0.117294, z_c, rx, ry, rz], a, v)
    movel(p[x_c + -0.043672, y_c + 0.117487, z_c, rx, ry, rz], a, v)
    movel(p[x_c + -0.043404, y_c + 0.117676, z_c, rx, ry, rz], a, v)
    movel(p[x_c + -0.043135, y_c + 0.117864, z_c, rx, ry, rz], a, v)
    movel(p[x_c + -0.042867, y_c + 0.118049, z_c, rx, ry, rz], a, v)
    movel(p[x_c + -0.042598, y_c + 0.118231, z_c, rx, ry, rz], a, v)
    movel(p[x_c + -0.042329, y_c + 0.118411, z_c, rx, ry, rz], a, v)
    movel(p[x_c + -0.042059, y_c + 0.118589, z_c, rx, ry, rz], a, v)
    movel(p[x_c + -0.041790, y_c + 0.118764, z_c, rx, ry, rz], a, v)
    movel(p[x_c + -0.041520, y_c + 0.118936, z_c, rx, ry, rz], a, v)
    movel(p[x_c + -0.041251, y_c + 0.119106, z_c, rx, ry, rz], a, v)
    movel(p[x_c + -0.040981, y_c + 0.119273, z_c, rx, ry, rz], a, v)
    movel(p[x_c + -0.040712, y_c + 0.119438, z_c, rx, ry, rz], a, v)
    movel(p[x_c + -0.040442, y_c + 0.119600, z_c, rx, ry, rz], a, v)
    movel(p[x_c + -0.040173, y_c + 0.119760, z_c, rx, ry, rz], a, v)
    movel(p[x_c + -0.039904, y_c + 0.119916, z_c, rx, ry, rz], a, v)
    movel(p[x_c + -0.039635, y_c + 0.120070, z_c, rx, ry, rz], a, v)
    movel(p[x_c + -0.039366, y_c + 0.120222, z_c, rx, ry, rz], a, v)
    movel(p[x_c + -0.039098, y_c + 0.120370, z_c, rx, ry, rz], a, v)
    movel(p[x_c + -0.038829, y_c + 0.120516, z_c, rx, ry, rz], a, v)
    movel(p[x_c + -0.038561, y_c + 0.120659, z_c, rx, ry, rz], a, v)
    movel(p[x_c + -0.038293, y_c + 0.120800, z_c, rx, ry, rz], a, v)
    movel(p[x_c + -0.038026, y_c + 0.120937, z_c, rx, ry, rz], a, v)
    movel(p[x_c + -0.037759, y_c + 0.121072, z_c, rx, ry, rz], a, v)
    movel(p[x_c + -0.037493, y_c + 0.121204, z_c, rx, ry, rz], a, v)
    movel(p[x_c + -0.037227, y_c + 0.121333, z_c, rx, ry, rz], a, v)
    movel(p[x_c + -0.036961, y_c + 0.121459, z_c, rx, ry, rz], a, v)
    movel(p[x_c + -0.036696, y_c + 0.121583, z_c, rx, ry, rz], a, v)
    movel(p[x_c + -0.036432, y_c + 0.121703, z_c, rx, ry, rz], a, v)
    movel(p[x_c + -0.036168, y_c + 0.121821, z_c, rx, ry, rz], a, v)
    movel(p[x_c + -0.035905, y_c + 0.121935, z_c, rx, ry, rz], a, v)
    movel(p[x_c + -0.035642, y_c + 0.122047, z_c, rx, ry, rz], a, v)
    movel(p[x_c + -0.035380, y_c + 0.122155, z_c, rx, ry, rz], a, v)
    movel(p[x_c + -0.035119, y_c + 0.122261, z_c, rx, ry, rz], a, v)
    movel(p[x_c + -0.034859, y_c + 0.122363, z_c, rx, ry, rz], a, v)
    movel(p[x_c + -0.034599, y_c + 0.122463, z_c, rx, ry, rz], a, v)
    movel(p[x_c + -0.034340, y_c + 0.122559, z_c, rx, ry, rz], a, v)
    movel(p[x_c + -0.034083, y_c + 0.122652, z_c, rx, ry, rz], a, v)
    movel(p[x_c + -0.033826, y_c + 0.122743, z_c, rx, ry, rz], a, v)
    movel(p[x_c + -0.033570, y_c + 0.122830, z_c, rx, ry, rz], a, v)
    movel(p[x_c + -0.033570, y_c + 0.122830, z_c, rx, ry, rz], a, v)
    movel(p[x_c + -0.033347, y_c + 0.122903, z_c, rx, ry, rz], a, v)
    movel(p[x_c + -0.033128, y_c + 0.122975, z_c, rx, ry, rz], a, v)
    movel(p[x_c + -0.032912, y_c + 0.123045, z_c, rx, ry, rz], a, v)
    movel(p[x_c + -0.032699, y_c + 0.123112, z_c, rx, ry, rz], a, v)
    movel(p[x_c + -0.032489, y_c + 0.123177, z_c, rx, ry, rz], a, v)
    movel(p[x_c + -0.032281, y_c + 0.123240, z_c, rx, ry, rz], a, v)
    movel(p[x_c + -0.032076, y_c + 0.123301, z_c, rx, ry, rz], a, v)
    movel(p[x_c + -0.031872, y_c + 0.123360, z_c, rx, ry, rz], a, v)
    movel(p[x_c + -0.031671, y_c + 0.123417, z_c, rx, ry, rz], a, v)
    movel(p[x_c + -0.031471, y_c + 0.123472, z_c, rx, ry, rz], a, v)
    movel(p[x_c + -0.031273, y_c + 0.123526, z_c, rx, ry, rz], a, v)
    movel(p[x_c + -0.031077, y_c + 0.123577, z_c, rx, ry, rz], a, v)
    movel(p[x_c + -0.030881, y_c + 0.123626, z_c, rx, ry, rz], a, v)
    movel(p[x_c + -0.030686, y_c + 0.123674, z_c, rx, ry, rz], a, v)
    movel(p[x_c + -0.030493, y_c + 0.123719, z_c, rx, ry, rz], a, v)
    movel(p[x_c + -0.030300, y_c + 0.123763, z_c, rx, ry, rz], a, v)
    movel(p[x_c + -0.030107, y_c + 0.123805, z_c, rx, ry, rz], a, v)
    movel(p[x_c + -0.029915, y_c + 0.123846, z_c, rx, ry, rz], a, v)
    movel(p[x_c + -0.029722, y_c + 0.123884, z_c, rx, ry, rz], a, v)
    movel(p[x_c + -0.029530, y_c + 0.123921, z_c, rx, ry, rz], a, v)
    movel(p[x_c + -0.029337, y_c + 0.123956, z_c, rx, ry, rz], a, v)
    movel(p[x_c + -0.029144, y_c + 0.123990, z_c, rx, ry, rz], a, v)
    movel(p[x_c + -0.028950, y_c + 0.124022, z_c, rx, ry, rz], a, v)
    movel(p[x_c + -0.028755, y_c + 0.124052, z_c, rx, ry, rz], a, v)
    movel(p[x_c + -0.028559, y_c + 0.124081, z_c, rx, ry, rz], a, v)
    movel(p[x_c + -0.028362, y_c + 0.124108, z_c, rx, ry, rz], a, v)
    movel(p[x_c + -0.028163, y_c + 0.124134, z_c, rx, ry, rz], a, v)
    movel(p[x_c + -0.027963, y_c + 0.124159, z_c, rx, ry, rz], a, v)
    movel(p[x_c + -0.027761, y_c + 0.124182, z_c, rx, ry, rz], a, v)
    movel(p[x_c + -0.027557, y_c + 0.124203, z_c, rx, ry, rz], a, v)
    movel(p[x_c + -0.027350, y_c + 0.124223, z_c, rx, ry, rz], a, v)
    movel(p[x_c + -0.027141, y_c + 0.124242, z_c, rx, ry, rz], a, v)
    movel(p[x_c + -0.026930, y_c + 0.124259, z_c, rx, ry, rz], a, v)
    movel(p[x_c + -0.026716, y_c + 0.124275, z_c, rx, ry, rz], a, v)
    movel(p[x_c + -0.026499, y_c + 0.124290, z_c, rx, ry, rz], a, v)
    movel(p[x_c + -0.026279, y_c + 0.124304, z_c, rx, ry, rz], a, v)
    movel(p[x_c + -0.026055, y_c + 0.124316, z_c, rx, ry, rz], a, v)
    movel(p[x_c + -0.025828, y_c + 0.124327, z_c, rx, ry, rz], a, v)
    movel(p[x_c + -0.025598, y_c + 0.124337, z_c, rx, ry, rz], a, v)
    movel(p[x_c + -0.025363, y_c + 0.124346, z_c, rx, ry, rz], a, v)
    movel(p[x_c + -0.025124, y_c + 0.124354, z_c, rx, ry, rz], a, v)
    movel(p[x_c + -0.024881, y_c + 0.124361, z_c, rx, ry, rz], a, v)
    movel(p[x_c + -0.024634, y_c + 0.124366, z_c, rx, ry, rz], a, v)
    movel(p[x_c + -0.024382, y_c + 0.124371, z_c, rx, ry, rz], a, v)
    movel(p[x_c + -0.024125, y_c + 0.124374, z_c, rx, ry, rz], a, v)
    movel(p[x_c + -0.023863, y_c + 0.124377, z_c, rx, ry, rz], a, v)
    movel(p[x_c + -0.023596, y_c + 0.124379, z_c, rx, ry, rz], a, v)
    movel(p[x_c + -0.023323, y_c + 0.124379, z_c, rx, ry, rz], a, v)
    movel(p[x_c + -0.023045, y_c + 0.124379, z_c, rx, ry, rz], a, v)
    movel(p[x_c + -0.023045, y_c + 0.124379, z_c, rx, ry, rz], a, v)
    movel(p[x_c + -0.022667, y_c + 0.124377, z_c, rx, ry, rz], a, v)
    movel(p[x_c + -0.022293, y_c + 0.124373, z_c, rx, ry, rz], a, v)
    movel(p[x_c + -0.021923, y_c + 0.124366, z_c, rx, ry, rz], a, v)
    movel(p[x_c + -0.021558, y_c + 0.124356, z_c, rx, ry, rz], a, v)
    movel(p[x_c + -0.021198, y_c + 0.124343, z_c, rx, ry, rz], a, v)
    movel(p[x_c + -0.020841, y_c + 0.124328, z_c, rx, ry, rz], a, v)
    movel(p[x_c + -0.020488, y_c + 0.124311, z_c, rx, ry, rz], a, v)
    movel(p[x_c + -0.020138, y_c + 0.124290, z_c, rx, ry, rz], a, v)
    movel(p[x_c + -0.019793, y_c + 0.124267, z_c, rx, ry, rz], a, v)
    movel(p[x_c + -0.019450, y_c + 0.124240, z_c, rx, ry, rz], a, v)
    movel(p[x_c + -0.019111, y_c + 0.124211, z_c, rx, ry, rz], a, v)
    movel(p[x_c + -0.018774, y_c + 0.124179, z_c, rx, ry, rz], a, v)
    movel(p[x_c + -0.018441, y_c + 0.124144, z_c, rx, ry, rz], a, v)
    movel(p[x_c + -0.018110, y_c + 0.124106, z_c, rx, ry, rz], a, v)
    movel(p[x_c + -0.017782, y_c + 0.124065, z_c, rx, ry, rz], a, v)
    movel(p[x_c + -0.017456, y_c + 0.124021, z_c, rx, ry, rz], a, v)
    movel(p[x_c + -0.017132, y_c + 0.123974, z_c, rx, ry, rz], a, v)
    movel(p[x_c + -0.016811, y_c + 0.123924, z_c, rx, ry, rz], a, v)
    movel(p[x_c + -0.016491, y_c + 0.123871, z_c, rx, ry, rz], a, v)
    movel(p[x_c + -0.016173, y_c + 0.123814, z_c, rx, ry, rz], a, v)
    movel(p[x_c + -0.015857, y_c + 0.123754, z_c, rx, ry, rz], a, v)
    movel(p[x_c + -0.015542, y_c + 0.123691, z_c, rx, ry, rz], a, v)
    movel(p[x_c + -0.015228, y_c + 0.123624, z_c, rx, ry, rz], a, v)
    movel(p[x_c + -0.014915, y_c + 0.123554, z_c, rx, ry, rz], a, v)
    movel(p[x_c + -0.014603, y_c + 0.123481, z_c, rx, ry, rz], a, v)
    movel(p[x_c + -0.014292, y_c + 0.123404, z_c, rx, ry, rz], a, v)
    movel(p[x_c + -0.013982, y_c + 0.123324, z_c, rx, ry, rz], a, v)
    movel(p[x_c + -0.013672, y_c + 0.123240, z_c, rx, ry, rz], a, v)
    movel(p[x_c + -0.013362, y_c + 0.123152, z_c, rx, ry, rz], a, v)
    movel(p[x_c + -0.013052, y_c + 0.123061, z_c, rx, ry, rz], a, v)
    movel(p[x_c + -0.012742, y_c + 0.122967, z_c, rx, ry, rz], a, v)
    movel(p[x_c + -0.012432, y_c + 0.122869, z_c, rx, ry, rz], a, v)
    movel(p[x_c + -0.012122, y_c + 0.122767, z_c, rx, ry, rz], a, v)
    movel(p[x_c + -0.011811, y_c + 0.122661, z_c, rx, ry, rz], a, v)
    movel(p[x_c + -0.011500, y_c + 0.122551, z_c, rx, ry, rz], a, v)
    movel(p[x_c + -0.011187, y_c + 0.122438, z_c, rx, ry, rz], a, v)
    movel(p[x_c + -0.010874, y_c + 0.122321, z_c, rx, ry, rz], a, v)
    movel(p[x_c + -0.010559, y_c + 0.122199, z_c, rx, ry, rz], a, v)
    movel(p[x_c + -0.010243, y_c + 0.122074, z_c, rx, ry, rz], a, v)
    movel(p[x_c + -0.009926, y_c + 0.121945, z_c, rx, ry, rz], a, v)
    movel(p[x_c + -0.009606, y_c + 0.121812, z_c, rx, ry, rz], a, v)
    movel(p[x_c + -0.009285, y_c + 0.121675, z_c, rx, ry, rz], a, v)
    movel(p[x_c + -0.008962, y_c + 0.121534, z_c, rx, ry, rz], a, v)
    movel(p[x_c + -0.008637, y_c + 0.121388, z_c, rx, ry, rz], a, v)
    movel(p[x_c + -0.008309, y_c + 0.121239, z_c, rx, ry, rz], a, v)
    movel(p[x_c + -0.007979, y_c + 0.121085, z_c, rx, ry, rz], a, v)
    movel(p[x_c + -0.007647, y_c + 0.120927, z_c, rx, ry, rz], a, v)
    movel(p[x_c + -0.007311, y_c + 0.120764, z_c, rx, ry, rz], a, v)
    movel(p[x_c + -0.006973, y_c + 0.120598, z_c, rx, ry, rz], a, v)
    movel(p[x_c + -0.006973, y_c + 0.120598, z_c, rx, ry, rz], a, v)
    movel(p[x_c + -0.006544, y_c + 0.120381, z_c, rx, ry, rz], a, v)
    movel(p[x_c + -0.006118, y_c + 0.120157, z_c, rx, ry, rz], a, v)
    movel(p[x_c + -0.005695, y_c + 0.119927, z_c, rx, ry, rz], a, v)
    movel(p[x_c + -0.005275, y_c + 0.119690, z_c, rx, ry, rz], a, v)
    movel(p[x_c + -0.004858, y_c + 0.119447, z_c, rx, ry, rz], a, v)
    movel(p[x_c + -0.004444, y_c + 0.119198, z_c, rx, ry, rz], a, v)
    movel(p[x_c + -0.004034, y_c + 0.118942, z_c, rx, ry, rz], a, v)
    movel(p[x_c + -0.003626, y_c + 0.118679, z_c, rx, ry, rz], a, v)
    movel(p[x_c + -0.003222, y_c + 0.118410, z_c, rx, ry, rz], a, v)
    movel(p[x_c + -0.002820, y_c + 0.118135, z_c, rx, ry, rz], a, v)
    movel(p[x_c + -0.002422, y_c + 0.117853, z_c, rx, ry, rz], a, v)
    movel(p[x_c + -0.002027, y_c + 0.117564, z_c, rx, ry, rz], a, v)
    movel(p[x_c + -0.001635, y_c + 0.117269, z_c, rx, ry, rz], a, v)
    movel(p[x_c + -0.001245, y_c + 0.116968, z_c, rx, ry, rz], a, v)
    movel(p[x_c + -0.000859, y_c + 0.116660, z_c, rx, ry, rz], a, v)
    movel(p[x_c + -0.000477, y_c + 0.116345, z_c, rx, ry, rz], a, v)
    movel(p[x_c + -0.000097, y_c + 0.116024, z_c, rx, ry, rz], a, v)
    movel(p[x_c + 0.000280, y_c + 0.115696, z_c, rx, ry, rz], a, v)
    movel(p[x_c + 0.000654, y_c + 0.115362, z_c, rx, ry, rz], a, v)
    movel(p[x_c + 0.001025, y_c + 0.115022, z_c, rx, ry, rz], a, v)
    movel(p[x_c + 0.001392, y_c + 0.114675, z_c, rx, ry, rz], a, v)
    movel(p[x_c + 0.001757, y_c + 0.114321, z_c, rx, ry, rz], a, v)
    movel(p[x_c + 0.002118, y_c + 0.113961, z_c, rx, ry, rz], a, v)
    movel(p[x_c + 0.002477, y_c + 0.113594, z_c, rx, ry, rz], a, v)
    movel(p[x_c + 0.002832, y_c + 0.113221, z_c, rx, ry, rz], a, v)
    movel(p[x_c + 0.003185, y_c + 0.112841, z_c, rx, ry, rz], a, v)
    movel(p[x_c + 0.003534, y_c + 0.112455, z_c, rx, ry, rz], a, v)
    movel(p[x_c + 0.003880, y_c + 0.112062, z_c, rx, ry, rz], a, v)
    movel(p[x_c + 0.004224, y_c + 0.111663, z_c, rx, ry, rz], a, v)
    movel(p[x_c + 0.004564, y_c + 0.111257, z_c, rx, ry, rz], a, v)
    movel(p[x_c + 0.004901, y_c + 0.110845, z_c, rx, ry, rz], a, v)
    movel(p[x_c + 0.005235, y_c + 0.110426, z_c, rx, ry, rz], a, v)
    movel(p[x_c + 0.005566, y_c + 0.110000, z_c, rx, ry, rz], a, v)
    movel(p[x_c + 0.005895, y_c + 0.109568, z_c, rx, ry, rz], a, v)
    movel(p[x_c + 0.006220, y_c + 0.109129, z_c, rx, ry, rz], a, v)
    movel(p[x_c + 0.006542, y_c + 0.108684, z_c, rx, ry, rz], a, v)
    movel(p[x_c + 0.006861, y_c + 0.108233, z_c, rx, ry, rz], a, v)
    movel(p[x_c + 0.007177, y_c + 0.107774, z_c, rx, ry, rz], a, v)
    movel(p[x_c + 0.007490, y_c + 0.107309, z_c, rx, ry, rz], a, v)
    movel(p[x_c + 0.007800, y_c + 0.106838, z_c, rx, ry, rz], a, v)
    movel(p[x_c + 0.008107, y_c + 0.106360, z_c, rx, ry, rz], a, v)
    movel(p[x_c + 0.008411, y_c + 0.105875, z_c, rx, ry, rz], a, v)
    movel(p[x_c + 0.008712, y_c + 0.105384, z_c, rx, ry, rz], a, v)
    movel(p[x_c + 0.009010, y_c + 0.104886, z_c, rx, ry, rz], a, v)
    movel(p[x_c + 0.009305, y_c + 0.104382, z_c, rx, ry, rz], a, v)
    movel(p[x_c + 0.009597, y_c + 0.103871, z_c, rx, ry, rz], a, v)
    movel(p[x_c + 0.009886, y_c + 0.103354, z_c, rx, ry, rz], a, v)
    movel(p[x_c + 0.010172, y_c + 0.102829, z_c, rx, ry, rz], a, v)
    movel(p[x_c + 0.010455, y_c + 0.102299, z_c, rx, ry, rz], a, v)
    movel(p[x_c + 0.010455, y_c + 0.102299, z_c, rx, ry, rz], a, v)
    movel(p[x_c + 0.010619, y_c + 0.101985, z_c, rx, ry, rz], a, v)
    movel(p[x_c + 0.010781, y_c + 0.101673, z_c, rx, ry, rz], a, v)
    movel(p[x_c + 0.010939, y_c + 0.101360, z_c, rx, ry, rz], a, v)
    movel(p[x_c + 0.011095, y_c + 0.101048, z_c, rx, ry, rz], a, v)
    movel(p[x_c + 0.011248, y_c + 0.100736, z_c, rx, ry, rz], a, v)
    movel(p[x_c + 0.011398, y_c + 0.100424, z_c, rx, ry, rz], a, v)
    movel(p[x_c + 0.011546, y_c + 0.100112, z_c, rx, ry, rz], a, v)
    movel(p[x_c + 0.011692, y_c + 0.099800, z_c, rx, ry, rz], a, v)
    movel(p[x_c + 0.011834, y_c + 0.099487, z_c, rx, ry, rz], a, v)
    movel(p[x_c + 0.011975, y_c + 0.099175, z_c, rx, ry, rz], a, v)
    movel(p[x_c + 0.012112, y_c + 0.098861, z_c, rx, ry, rz], a, v)
    movel(p[x_c + 0.012248, y_c + 0.098547, z_c, rx, ry, rz], a, v)
    movel(p[x_c + 0.012381, y_c + 0.098233, z_c, rx, ry, rz], a, v)
    movel(p[x_c + 0.012512, y_c + 0.097917, z_c, rx, ry, rz], a, v)
    movel(p[x_c + 0.012640, y_c + 0.097601, z_c, rx, ry, rz], a, v)
    movel(p[x_c + 0.012766, y_c + 0.097283, z_c, rx, ry, rz], a, v)
    movel(p[x_c + 0.012890, y_c + 0.096964, z_c, rx, ry, rz], a, v)
    movel(p[x_c + 0.013012, y_c + 0.096644, z_c, rx, ry, rz], a, v)
    movel(p[x_c + 0.013131, y_c + 0.096323, z_c, rx, ry, rz], a, v)
    movel(p[x_c + 0.013249, y_c + 0.096000, z_c, rx, ry, rz], a, v)
    movel(p[x_c + 0.013364, y_c + 0.095676, z_c, rx, ry, rz], a, v)
    movel(p[x_c + 0.013477, y_c + 0.095349, z_c, rx, ry, rz], a, v)
    movel(p[x_c + 0.013588, y_c + 0.095021, z_c, rx, ry, rz], a, v)
    movel(p[x_c + 0.013698, y_c + 0.094691, z_c, rx, ry, rz], a, v)
    movel(p[x_c + 0.013805, y_c + 0.094359, z_c, rx, ry, rz], a, v)
    movel(p[x_c + 0.013910, y_c + 0.094025, z_c, rx, ry, rz], a, v)
    movel(p[x_c + 0.014014, y_c + 0.093688, z_c, rx, ry, rz], a, v)
    movel(p[x_c + 0.014115, y_c + 0.093349, z_c, rx, ry, rz], a, v)
    movel(p[x_c + 0.014215, y_c + 0.093008, z_c, rx, ry, rz], a, v)
    movel(p[x_c + 0.014313, y_c + 0.092663, z_c, rx, ry, rz], a, v)
    movel(p[x_c + 0.014410, y_c + 0.092316, z_c, rx, ry, rz], a, v)
    movel(p[x_c + 0.014504, y_c + 0.091967, z_c, rx, ry, rz], a, v)
    movel(p[x_c + 0.014597, y_c + 0.091614, z_c, rx, ry, rz], a, v)
    movel(p[x_c + 0.014689, y_c + 0.091258, z_c, rx, ry, rz], a, v)
    movel(p[x_c + 0.014779, y_c + 0.090899, z_c, rx, ry, rz], a, v)
    movel(p[x_c + 0.014867, y_c + 0.090537, z_c, rx, ry, rz], a, v)
    movel(p[x_c + 0.014954, y_c + 0.090171, z_c, rx, ry, rz], a, v)
    movel(p[x_c + 0.015039, y_c + 0.089802, z_c, rx, ry, rz], a, v)
    movel(p[x_c + 0.015123, y_c + 0.089429, z_c, rx, ry, rz], a, v)
    movel(p[x_c + 0.015205, y_c + 0.089052, z_c, rx, ry, rz], a, v)
    movel(p[x_c + 0.015286, y_c + 0.088672, z_c, rx, ry, rz], a, v)
    movel(p[x_c + 0.015366, y_c + 0.088287, z_c, rx, ry, rz], a, v)
    movel(p[x_c + 0.015444, y_c + 0.087899, z_c, rx, ry, rz], a, v)
    movel(p[x_c + 0.015522, y_c + 0.087506, z_c, rx, ry, rz], a, v)
    movel(p[x_c + 0.015598, y_c + 0.087109, z_c, rx, ry, rz], a, v)
    movel(p[x_c + 0.015672, y_c + 0.086707, z_c, rx, ry, rz], a, v)
    movel(p[x_c + 0.015746, y_c + 0.086301, z_c, rx, ry, rz], a, v)
    movel(p[x_c + 0.015818, y_c + 0.085890, z_c, rx, ry, rz], a, v)
    movel(p[x_c + 0.015890, y_c + 0.085475, z_c, rx, ry, rz], a, v)
    movel(p[x_c + 0.015890, y_c + 0.085475, z_c, rx, ry, rz], a, v)
    movel(p[x_c + 0.015959, y_c + 0.085070, z_c, rx, ry, rz], a, v)
    movel(p[x_c + 0.016027, y_c + 0.084677, z_c, rx, ry, rz], a, v)
    movel(p[x_c + 0.016095, y_c + 0.084296, z_c, rx, ry, rz], a, v)
    movel(p[x_c + 0.016162, y_c + 0.083927, z_c, rx, ry, rz], a, v)
    movel(p[x_c + 0.016228, y_c + 0.083569, z_c, rx, ry, rz], a, v)
    movel(p[x_c + 0.016295, y_c + 0.083222, z_c, rx, ry, rz], a, v)
    movel(p[x_c + 0.016361, y_c + 0.082885, z_c, rx, ry, rz], a, v)
    movel(p[x_c + 0.016427, y_c + 0.082558, z_c, rx, ry, rz], a, v)
    movel(p[x_c + 0.016494, y_c + 0.082241, z_c, rx, ry, rz], a, v)
    movel(p[x_c + 0.016561, y_c + 0.081932, z_c, rx, ry, rz], a, v)
    movel(p[x_c + 0.016629, y_c + 0.081632, z_c, rx, ry, rz], a, v)
    movel(p[x_c + 0.016697, y_c + 0.081341, z_c, rx, ry, rz], a, v)
    movel(p[x_c + 0.016767, y_c + 0.081057, z_c, rx, ry, rz], a, v)
    movel(p[x_c + 0.016838, y_c + 0.080780, z_c, rx, ry, rz], a, v)
    movel(p[x_c + 0.016910, y_c + 0.080511, z_c, rx, ry, rz], a, v)
    movel(p[x_c + 0.016984, y_c + 0.080248, z_c, rx, ry, rz], a, v)
    movel(p[x_c + 0.017059, y_c + 0.079991, z_c, rx, ry, rz], a, v)
    movel(p[x_c + 0.017137, y_c + 0.079740, z_c, rx, ry, rz], a, v)
    movel(p[x_c + 0.017216, y_c + 0.079495, z_c, rx, ry, rz], a, v)
    movel(p[x_c + 0.017298, y_c + 0.079254, z_c, rx, ry, rz], a, v)
    movel(p[x_c + 0.017382, y_c + 0.079017, z_c, rx, ry, rz], a, v)
    movel(p[x_c + 0.017469, y_c + 0.078785, z_c, rx, ry, rz], a, v)
    movel(p[x_c + 0.017559, y_c + 0.078556, z_c, rx, ry, rz], a, v)
    movel(p[x_c + 0.017651, y_c + 0.078331, z_c, rx, ry, rz], a, v)
    movel(p[x_c + 0.017747, y_c + 0.078108, z_c, rx, ry, rz], a, v)
    movel(p[x_c + 0.017846, y_c + 0.077888, z_c, rx, ry, rz], a, v)
    movel(p[x_c + 0.017949, y_c + 0.077670, z_c, rx, ry, rz], a, v)
    movel(p[x_c + 0.018056, y_c + 0.077453, z_c, rx, ry, rz], a, v)
    movel(p[x_c + 0.018166, y_c + 0.077237, z_c, rx, ry, rz], a, v)
    movel(p[x_c + 0.018280, y_c + 0.077022, z_c, rx, ry, rz], a, v)
    movel(p[x_c + 0.018399, y_c + 0.076808, z_c, rx, ry, rz], a, v)
    movel(p[x_c + 0.018522, y_c + 0.076593, z_c, rx, ry, rz], a, v)
    movel(p[x_c + 0.018650, y_c + 0.076378, z_c, rx, ry, rz], a, v)
    movel(p[x_c + 0.018782, y_c + 0.076161, z_c, rx, ry, rz], a, v)
    movel(p[x_c + 0.018920, y_c + 0.075944, z_c, rx, ry, rz], a, v)
    movel(p[x_c + 0.019062, y_c + 0.075724, z_c, rx, ry, rz], a, v)
    movel(p[x_c + 0.019210, y_c + 0.075503, z_c, rx, ry, rz], a, v)
    movel(p[x_c + 0.019364, y_c + 0.075278, z_c, rx, ry, rz], a, v)
    movel(p[x_c + 0.019523, y_c + 0.075051, z_c, rx, ry, rz], a, v)
    movel(p[x_c + 0.019688, y_c + 0.074820, z_c, rx, ry, rz], a, v)
    movel(p[x_c + 0.019859, y_c + 0.074586, z_c, rx, ry, rz], a, v)
    movel(p[x_c + 0.020036, y_c + 0.074347, z_c, rx, ry, rz], a, v)
    movel(p[x_c + 0.020220, y_c + 0.074103, z_c, rx, ry, rz], a, v)
    movel(p[x_c + 0.020410, y_c + 0.073854, z_c, rx, ry, rz], a, v)
    movel(p[x_c + 0.020607, y_c + 0.073600, z_c, rx, ry, rz], a, v)
    movel(p[x_c + 0.020811, y_c + 0.073339, z_c, rx, ry, rz], a, v)
    movel(p[x_c + 0.021022, y_c + 0.073073, z_c, rx, ry, rz], a, v)
    movel(p[x_c + 0.021241, y_c + 0.072799, z_c, rx, ry, rz], a, v)
    movel(p[x_c + 0.021467, y_c + 0.072518, z_c, rx, ry, rz], a, v)
    movel(p[x_c + 0.021467, y_c + 0.072518, z_c, rx, ry, rz], a, v)
    movel(p[x_c + 0.022159, y_c + 0.071654, z_c, rx, ry, rz], a, v)
    movel(p[x_c + 0.022848, y_c + 0.070781, z_c, rx, ry, rz], a, v)
    movel(p[x_c + 0.023532, y_c + 0.069902, z_c, rx, ry, rz], a, v)
    movel(p[x_c + 0.024212, y_c + 0.069014, z_c, rx, ry, rz], a, v)
    movel(p[x_c + 0.024888, y_c + 0.068120, z_c, rx, ry, rz], a, v)
    movel(p[x_c + 0.025558, y_c + 0.067218, z_c, rx, ry, rz], a, v)
    movel(p[x_c + 0.026224, y_c + 0.066310, z_c, rx, ry, rz], a, v)
    movel(p[x_c + 0.026885, y_c + 0.065396, z_c, rx, ry, rz], a, v)
    movel(p[x_c + 0.027541, y_c + 0.064475, z_c, rx, ry, rz], a, v)
    movel(p[x_c + 0.028192, y_c + 0.063548, z_c, rx, ry, rz], a, v)
    movel(p[x_c + 0.028837, y_c + 0.062615, z_c, rx, ry, rz], a, v)
    movel(p[x_c + 0.029478, y_c + 0.061676, z_c, rx, ry, rz], a, v)
    movel(p[x_c + 0.030112, y_c + 0.060732, z_c, rx, ry, rz], a, v)
    movel(p[x_c + 0.030741, y_c + 0.059783, z_c, rx, ry, rz], a, v)
    movel(p[x_c + 0.031365, y_c + 0.058829, z_c, rx, ry, rz], a, v)
    movel(p[x_c + 0.031982, y_c + 0.057870, z_c, rx, ry, rz], a, v)
    movel(p[x_c + 0.032594, y_c + 0.056907, z_c, rx, ry, rz], a, v)
    movel(p[x_c + 0.033199, y_c + 0.055939, z_c, rx, ry, rz], a, v)
    movel(p[x_c + 0.033798, y_c + 0.054966, z_c, rx, ry, rz], a, v)
    movel(p[x_c + 0.034391, y_c + 0.053990, z_c, rx, ry, rz], a, v)
    movel(p[x_c + 0.034977, y_c + 0.053011, z_c, rx, ry, rz], a, v)
    movel(p[x_c + 0.035557, y_c + 0.052027, z_c, rx, ry, rz], a, v)
    movel(p[x_c + 0.036130, y_c + 0.051041, z_c, rx, ry, rz], a, v)
    movel(p[x_c + 0.036696, y_c + 0.050051, z_c, rx, ry, rz], a, v)
    movel(p[x_c + 0.037256, y_c + 0.049058, z_c, rx, ry, rz], a, v)
    movel(p[x_c + 0.037808, y_c + 0.048063, z_c, rx, ry, rz], a, v)
    movel(p[x_c + 0.038353, y_c + 0.047065, z_c, rx, ry, rz], a, v)
    movel(p[x_c + 0.038891, y_c + 0.046065, z_c, rx, ry, rz], a, v)
    movel(p[x_c + 0.039421, y_c + 0.045063, z_c, rx, ry, rz], a, v)
    movel(p[x_c + 0.039944, y_c + 0.044059, z_c, rx, ry, rz], a, v)
    movel(p[x_c + 0.040459, y_c + 0.043054, z_c, rx, ry, rz], a, v)
    movel(p[x_c + 0.040966, y_c + 0.042047, z_c, rx, ry, rz], a, v)
    movel(p[x_c + 0.041466, y_c + 0.041039, z_c, rx, ry, rz], a, v)
    movel(p[x_c + 0.041957, y_c + 0.040030, z_c, rx, ry, rz], a, v)
    movel(p[x_c + 0.042440, y_c + 0.039020, z_c, rx, ry, rz], a, v)
    movel(p[x_c + 0.042915, y_c + 0.038010, z_c, rx, ry, rz], a, v)
    movel(p[x_c + 0.043382, y_c + 0.036999, z_c, rx, ry, rz], a, v)
    movel(p[x_c + 0.043840, y_c + 0.035989, z_c, rx, ry, rz], a, v)
    movel(p[x_c + 0.044289, y_c + 0.034978, z_c, rx, ry, rz], a, v)
    movel(p[x_c + 0.044730, y_c + 0.033968, z_c, rx, ry, rz], a, v)
    movel(p[x_c + 0.045162, y_c + 0.032958, z_c, rx, ry, rz], a, v)
    movel(p[x_c + 0.045585, y_c + 0.031949, z_c, rx, ry, rz], a, v)
    movel(p[x_c + 0.045999, y_c + 0.030941, z_c, rx, ry, rz], a, v)
    movel(p[x_c + 0.046403, y_c + 0.029934, z_c, rx, ry, rz], a, v)
    movel(p[x_c + 0.046798, y_c + 0.028928, z_c, rx, ry, rz], a, v)
    movel(p[x_c + 0.047184, y_c + 0.027924, z_c, rx, ry, rz], a, v)
    movel(p[x_c + 0.047560, y_c + 0.026922, z_c, rx, ry, rz], a, v)
    movel(p[x_c + 0.047927, y_c + 0.025921, z_c, rx, ry, rz], a, v)
    movel(p[x_c + 0.048284, y_c + 0.024923, z_c, rx, ry, rz], a, v)
    movel(p[x_c + 0.048284, y_c + 0.024923, z_c, rx, ry, rz], a, v)
    movel(p[x_c + 0.048647, y_c + 0.023881, z_c, rx, ry, rz], a, v)
    movel(p[x_c + 0.049006, y_c + 0.022826, z_c, rx, ry, rz], a, v)
    movel(p[x_c + 0.049362, y_c + 0.021756, z_c, rx, ry, rz], a, v)
    movel(p[x_c + 0.049713, y_c + 0.020674, z_c, rx, ry, rz], a, v)
    movel(p[x_c + 0.050061, y_c + 0.019579, z_c, rx, ry, rz], a, v)
    movel(p[x_c + 0.050404, y_c + 0.018472, z_c, rx, ry, rz], a, v)
    movel(p[x_c + 0.050743, y_c + 0.017354, z_c, rx, ry, rz], a, v)
    movel(p[x_c + 0.051078, y_c + 0.016224, z_c, rx, ry, rz], a, v)
    movel(p[x_c + 0.051408, y_c + 0.015084, z_c, rx, ry, rz], a, v)
    movel(p[x_c + 0.051734, y_c + 0.013933, z_c, rx, ry, rz], a, v)
    movel(p[x_c + 0.052055, y_c + 0.012773, z_c, rx, ry, rz], a, v)
    movel(p[x_c + 0.052371, y_c + 0.011603, z_c, rx, ry, rz], a, v)
    movel(p[x_c + 0.052683, y_c + 0.010425, z_c, rx, ry, rz], a, v)
    movel(p[x_c + 0.052990, y_c + 0.009239, z_c, rx, ry, rz], a, v)
    movel(p[x_c + 0.053291, y_c + 0.008044, z_c, rx, ry, rz], a, v)
    movel(p[x_c + 0.053588, y_c + 0.006842, z_c, rx, ry, rz], a, v)
    movel(p[x_c + 0.053879, y_c + 0.005634, z_c, rx, ry, rz], a, v)
    movel(p[x_c + 0.054165, y_c + 0.004418, z_c, rx, ry, rz], a, v)
    movel(p[x_c + 0.054446, y_c + 0.003197, z_c, rx, ry, rz], a, v)
    movel(p[x_c + 0.054721, y_c + 0.001971, z_c, rx, ry, rz], a, v)
    movel(p[x_c + 0.054991, y_c + 0.000739, z_c, rx, ry, rz], a, v)
    movel(p[x_c + 0.055255, y_c + -0.000497, z_c, rx, ry, rz], a, v)
    movel(p[x_c + 0.055513, y_c + -0.001738, z_c, rx, ry, rz], a, v)
    movel(p[x_c + 0.055765, y_c + -0.002981, z_c, rx, ry, rz], a, v)
    movel(p[x_c + 0.056012, y_c + -0.004229, z_c, rx, ry, rz], a, v)
    movel(p[x_c + 0.056252, y_c + -0.005478, z_c, rx, ry, rz], a, v)
    movel(p[x_c + 0.056487, y_c + -0.006730, z_c, rx, ry, rz], a, v)
    movel(p[x_c + 0.056715, y_c + -0.007984, z_c, rx, ry, rz], a, v)
    movel(p[x_c + 0.056937, y_c + -0.009239, z_c, rx, ry, rz], a, v)
    movel(p[x_c + 0.057152, y_c + -0.010495, z_c, rx, ry, rz], a, v)
    movel(p[x_c + 0.057361, y_c + -0.011751, z_c, rx, ry, rz], a, v)
    movel(p[x_c + 0.057564, y_c + -0.013007, z_c, rx, ry, rz], a, v)
    movel(p[x_c + 0.057759, y_c + -0.014263, z_c, rx, ry, rz], a, v)
    movel(p[x_c + 0.057948, y_c + -0.015517, z_c, rx, ry, rz], a, v)
    movel(p[x_c + 0.058130, y_c + -0.016770, z_c, rx, ry, rz], a, v)
    movel(p[x_c + 0.058306, y_c + -0.018020, z_c, rx, ry, rz], a, v)
    movel(p[x_c + 0.058474, y_c + -0.019269, z_c, rx, ry, rz], a, v)
    movel(p[x_c + 0.058635, y_c + -0.020514, z_c, rx, ry, rz], a, v)
    movel(p[x_c + 0.058788, y_c + -0.021756, z_c, rx, ry, rz], a, v)
    movel(p[x_c + 0.058935, y_c + -0.022994, z_c, rx, ry, rz], a, v)
    movel(p[x_c + 0.059074, y_c + -0.024228, z_c, rx, ry, rz], a, v)
    movel(p[x_c + 0.059205, y_c + -0.025457, z_c, rx, ry, rz], a, v)
    movel(p[x_c + 0.059329, y_c + -0.026681, z_c, rx, ry, rz], a, v)
    movel(p[x_c + 0.059445, y_c + -0.027898, z_c, rx, ry, rz], a, v)
    movel(p[x_c + 0.059554, y_c + -0.029110, z_c, rx, ry, rz], a, v)
    movel(p[x_c + 0.059654, y_c + -0.030315, z_c, rx, ry, rz], a, v)
    movel(p[x_c + 0.059747, y_c + -0.031513, z_c, rx, ry, rz], a, v)
    movel(p[x_c + 0.059831, y_c + -0.032703, z_c, rx, ry, rz], a, v)
    movel(p[x_c + 0.059908, y_c + -0.033885, z_c, rx, ry, rz], a, v)
    movel(p[x_c + 0.059908, y_c + -0.033885, z_c, rx, ry, rz], a, v)
    movel(p[x_c + 0.059927, y_c + -0.034221, z_c, rx, ry, rz], a, v)
    movel(p[x_c + 0.059945, y_c + -0.034581, z_c, rx, ry, rz], a, v)
    movel(p[x_c + 0.059962, y_c + -0.034964, z_c, rx, ry, rz], a, v)
    movel(p[x_c + 0.059977, y_c + -0.035368, z_c, rx, ry, rz], a, v)
    movel(p[x_c + 0.059991, y_c + -0.035792, z_c, rx, ry, rz], a, v)
    movel(p[x_c + 0.060004, y_c + -0.036236, z_c, rx, ry, rz], a, v)
    movel(p[x_c + 0.060016, y_c + -0.036699, z_c, rx, ry, rz], a, v)
    movel(p[x_c + 0.060027, y_c + -0.037179, z_c, rx, ry, rz], a, v)
    movel(p[x_c + 0.060036, y_c + -0.037676, z_c, rx, ry, rz], a, v)
    movel(p[x_c + 0.060044, y_c + -0.038189, z_c, rx, ry, rz], a, v)
    movel(p[x_c + 0.060051, y_c + -0.038716, z_c, rx, ry, rz], a, v)
    movel(p[x_c + 0.060057, y_c + -0.039258, z_c, rx, ry, rz], a, v)
    movel(p[x_c + 0.060061, y_c + -0.039812, z_c, rx, ry, rz], a, v)
    movel(p[x_c + 0.060065, y_c + -0.040379, z_c, rx, ry, rz], a, v)
    movel(p[x_c + 0.060067, y_c + -0.040956, z_c, rx, ry, rz], a, v)
    movel(p[x_c + 0.060069, y_c + -0.041544, z_c, rx, ry, rz], a, v)
    movel(p[x_c + 0.060069, y_c + -0.042141, z_c, rx, ry, rz], a, v)
    movel(p[x_c + 0.060068, y_c + -0.042746, z_c, rx, ry, rz], a, v)
    movel(p[x_c + 0.060066, y_c + -0.043359, z_c, rx, ry, rz], a, v)
    movel(p[x_c + 0.060063, y_c + -0.043978, z_c, rx, ry, rz], a, v)
    movel(p[x_c + 0.060059, y_c + -0.044602, z_c, rx, ry, rz], a, v)
    movel(p[x_c + 0.060054, y_c + -0.045231, z_c, rx, ry, rz], a, v)
    movel(p[x_c + 0.060048, y_c + -0.045863, z_c, rx, ry, rz], a, v)
    movel(p[x_c + 0.060041, y_c + -0.046498, z_c, rx, ry, rz], a, v)
    movel(p[x_c + 0.060032, y_c + -0.047134, z_c, rx, ry, rz], a, v)
    movel(p[x_c + 0.060023, y_c + -0.047771, z_c, rx, ry, rz], a, v)
    movel(p[x_c + 0.060013, y_c + -0.048408, z_c, rx, ry, rz], a, v)
    movel(p[x_c + 0.060002, y_c + -0.049044, z_c, rx, ry, rz], a, v)
    movel(p[x_c + 0.059990, y_c + -0.049678, z_c, rx, ry, rz], a, v)
    movel(p[x_c + 0.059977, y_c + -0.050308, z_c, rx, ry, rz], a, v)
    movel(p[x_c + 0.059963, y_c + -0.050935, z_c, rx, ry, rz], a, v)
    movel(p[x_c + 0.059948, y_c + -0.051556, z_c, rx, ry, rz], a, v)
    movel(p[x_c + 0.059933, y_c + -0.052172, z_c, rx, ry, rz], a, v)
    movel(p[x_c + 0.059916, y_c + -0.052781, z_c, rx, ry, rz], a, v)
    movel(p[x_c + 0.059898, y_c + -0.053382, z_c, rx, ry, rz], a, v)
    movel(p[x_c + 0.059880, y_c + -0.053974, z_c, rx, ry, rz], a, v)
    movel(p[x_c + 0.059861, y_c + -0.054557, z_c, rx, ry, rz], a, v)
    movel(p[x_c + 0.059841, y_c + -0.055129, z_c, rx, ry, rz], a, v)
    movel(p[x_c + 0.059820, y_c + -0.055689, z_c, rx, ry, rz], a, v)
    movel(p[x_c + 0.059798, y_c + -0.056237, z_c, rx, ry, rz], a, v)
    movel(p[x_c + 0.059775, y_c + -0.056771, z_c, rx, ry, rz], a, v)
    movel(p[x_c + 0.059752, y_c + -0.057291, z_c, rx, ry, rz], a, v)
    movel(p[x_c + 0.059728, y_c + -0.057796, z_c, rx, ry, rz], a, v)
    movel(p[x_c + 0.059703, y_c + -0.058285, z_c, rx, ry, rz], a, v)
    movel(p[x_c + 0.059677, y_c + -0.058756, z_c, rx, ry, rz], a, v)
    movel(p[x_c + 0.059651, y_c + -0.059209, z_c, rx, ry, rz], a, v)
    movel(p[x_c + 0.059624, y_c + -0.059643, z_c, rx, ry, rz], a, v)
    movel(p[x_c + 0.059596, y_c + -0.060056, z_c, rx, ry, rz], a, v)
    movel(p[x_c + 0.059567, y_c + -0.060449, z_c, rx, ry, rz], a, v)
    movel(p[x_c + 0.059567, y_c + -0.060449, z_c, rx, ry, rz], a, v)
    movel(p[x_c + 0.059556, y_c + -0.060603, z_c, rx, ry, rz], a, v)
    movel(p[x_c + 0.059544, y_c + -0.060762, z_c, rx, ry, rz], a, v)
    movel(p[x_c + 0.059532, y_c + -0.060927, z_c, rx, ry, rz], a, v)
    movel(p[x_c + 0.059519, y_c + -0.061097, z_c, rx, ry, rz], a, v)
    movel(p[x_c + 0.059507, y_c + -0.061273, z_c, rx, ry, rz], a, v)
    movel(p[x_c + 0.059494, y_c + -0.061453, z_c, rx, ry, rz], a, v)
    movel(p[x_c + 0.059480, y_c + -0.061639, z_c, rx, ry, rz], a, v)
    movel(p[x_c + 0.059467, y_c + -0.061829, z_c, rx, ry, rz], a, v)
    movel(p[x_c + 0.059453, y_c + -0.062024, z_c, rx, ry, rz], a, v)
    movel(p[x_c + 0.059439, y_c + -0.062223, z_c, rx, ry, rz], a, v)
    movel(p[x_c + 0.059425, y_c + -0.062426, z_c, rx, ry, rz], a, v)
    movel(p[x_c + 0.059411, y_c + -0.062633, z_c, rx, ry, rz], a, v)
    movel(p[x_c + 0.059397, y_c + -0.062843, z_c, rx, ry, rz], a, v)
    movel(p[x_c + 0.059382, y_c + -0.063058, z_c, rx, ry, rz], a, v)
    movel(p[x_c + 0.059367, y_c + -0.063275, z_c, rx, ry, rz], a, v)
    movel(p[x_c + 0.059353, y_c + -0.063496, z_c, rx, ry, rz], a, v)
    movel(p[x_c + 0.059338, y_c + -0.063720, z_c, rx, ry, rz], a, v)
    movel(p[x_c + 0.059323, y_c + -0.063946, z_c, rx, ry, rz], a, v)
    movel(p[x_c + 0.059307, y_c + -0.064175, z_c, rx, ry, rz], a, v)
    movel(p[x_c + 0.059292, y_c + -0.064406, z_c, rx, ry, rz], a, v)
    movel(p[x_c + 0.059277, y_c + -0.064640, z_c, rx, ry, rz], a, v)
    movel(p[x_c + 0.059261, y_c + -0.064875, z_c, rx, ry, rz], a, v)
    movel(p[x_c + 0.059246, y_c + -0.065113, z_c, rx, ry, rz], a, v)
    movel(p[x_c + 0.059231, y_c + -0.065352, z_c, rx, ry, rz], a, v)
    movel(p[x_c + 0.059215, y_c + -0.065592, z_c, rx, ry, rz], a, v)
    movel(p[x_c + 0.059200, y_c + -0.065833, z_c, rx, ry, rz], a, v)
    movel(p[x_c + 0.059184, y_c + -0.066076, z_c, rx, ry, rz], a, v)
    movel(p[x_c + 0.059169, y_c + -0.066319, z_c, rx, ry, rz], a, v)
    movel(p[x_c + 0.059153, y_c + -0.066563, z_c, rx, ry, rz], a, v)
    movel(p[x_c + 0.059138, y_c + -0.066807, z_c, rx, ry, rz], a, v)
    movel(p[x_c + 0.059123, y_c + -0.067052, z_c, rx, ry, rz], a, v)
    movel(p[x_c + 0.059107, y_c + -0.067297, z_c, rx, ry, rz], a, v)
    movel(p[x_c + 0.059092, y_c + -0.067541, z_c, rx, ry, rz], a, v)
    movel(p[x_c + 0.059077, y_c + -0.067785, z_c, rx, ry, rz], a, v)
    movel(p[x_c + 0.059062, y_c + -0.068029, z_c, rx, ry, rz], a, v)
    movel(p[x_c + 0.059047, y_c + -0.068272, z_c, rx, ry, rz], a, v)
    movel(p[x_c + 0.059033, y_c + -0.068514, z_c, rx, ry, rz], a, v)
    movel(p[x_c + 0.059018, y_c + -0.068755, z_c, rx, ry, rz], a, v)
    movel(p[x_c + 0.059004, y_c + -0.068995, z_c, rx, ry, rz], a, v)
    movel(p[x_c + 0.058989, y_c + -0.069233, z_c, rx, ry, rz], a, v)
    movel(p[x_c + 0.058975, y_c + -0.069469, z_c, rx, ry, rz], a, v)
    movel(p[x_c + 0.058961, y_c + -0.069704, z_c, rx, ry, rz], a, v)
    movel(p[x_c + 0.058948, y_c + -0.069936, z_c, rx, ry, rz], a, v)
    movel(p[x_c + 0.058934, y_c + -0.070166, z_c, rx, ry, rz], a, v)
    movel(p[x_c + 0.058921, y_c + -0.070394, z_c, rx, ry, rz], a, v)
    movel(p[x_c + 0.058908, y_c + -0.070619, z_c, rx, ry, rz], a, v)
    movel(p[x_c + 0.058895, y_c + -0.070841, z_c, rx, ry, rz], a, v)
    movel(p[x_c + 0.058883, y_c + -0.071060, z_c, rx, ry, rz], a, v)
    movel(p[x_c + 0.058871, y_c + -0.071276, z_c, rx, ry, rz], a, v)
    movel(p[x_c + 0.058871, y_c + -0.071276, z_c, rx, ry, rz], a, v)
    movel(p[x_c + 0.058826, y_c + -0.072092, z_c, rx, ry, rz], a, v)
    movel(p[x_c + 0.058787, y_c + -0.072881, z_c, rx, ry, rz], a, v)
    movel(p[x_c + 0.058753, y_c + -0.073643, z_c, rx, ry, rz], a, v)
    movel(p[x_c + 0.058725, y_c + -0.074380, z_c, rx, ry, rz], a, v)
    movel(p[x_c + 0.058703, y_c + -0.075092, z_c, rx, ry, rz], a, v)
    movel(p[x_c + 0.058688, y_c + -0.075780, z_c, rx, ry, rz], a, v)
    movel(p[x_c + 0.058681, y_c + -0.076446, z_c, rx, ry, rz], a, v)
    movel(p[x_c + 0.058681, y_c + -0.077091, z_c, rx, ry, rz], a, v)
    movel(p[x_c + 0.058690, y_c + -0.077715, z_c, rx, ry, rz], a, v)
    movel(p[x_c + 0.058708, y_c + -0.078320, z_c, rx, ry, rz], a, v)
    movel(p[x_c + 0.058735, y_c + -0.078907, z_c, rx, ry, rz], a, v)
    movel(p[x_c + 0.058772, y_c + -0.079476, z_c, rx, ry, rz], a, v)
    movel(p[x_c + 0.058819, y_c + -0.080029, z_c, rx, ry, rz], a, v)
    movel(p[x_c + 0.058877, y_c + -0.080567, z_c, rx, ry, rz], a, v)
    movel(p[x_c + 0.058946, y_c + -0.081090, z_c, rx, ry, rz], a, v)
    movel(p[x_c + 0.059027, y_c + -0.081600, z_c, rx, ry, rz], a, v)
    movel(p[x_c + 0.059120, y_c + -0.082098, z_c, rx, ry, rz], a, v)
    movel(p[x_c + 0.059226, y_c + -0.082584, z_c, rx, ry, rz], a, v)
    movel(p[x_c + 0.059345, y_c + -0.083061, z_c, rx, ry, rz], a, v)
    movel(p[x_c + 0.059478, y_c + -0.083528, z_c, rx, ry, rz], a, v)
    movel(p[x_c + 0.059625, y_c + -0.083987, z_c, rx, ry, rz], a, v)
    movel(p[x_c + 0.059786, y_c + -0.084438, z_c, rx, ry, rz], a, v)
    movel(p[x_c + 0.059963, y_c + -0.084884, z_c, rx, ry, rz], a, v)
    movel(p[x_c + 0.060156, y_c + -0.085324, z_c, rx, ry, rz], a, v)
    movel(p[x_c + 0.060365, y_c + -0.085761, z_c, rx, ry, rz], a, v)
    movel(p[x_c + 0.060590, y_c + -0.086194, z_c, rx, ry, rz], a, v)
    movel(p[x_c + 0.060832, y_c + -0.086625, z_c, rx, ry, rz], a, v)
    movel(p[x_c + 0.061092, y_c + -0.087055, z_c, rx, ry, rz], a, v)
    movel(p[x_c + 0.061371, y_c + -0.087486, z_c, rx, ry, rz], a, v)
    movel(p[x_c + 0.061667, y_c + -0.087917, z_c, rx, ry, rz], a, v)
    movel(p[x_c + 0.061983, y_c + -0.088350, z_c, rx, ry, rz], a, v)
    movel(p[x_c + 0.062319, y_c + -0.088786, z_c, rx, ry, rz], a, v)
    movel(p[x_c + 0.062674, y_c + -0.089226, z_c, rx, ry, rz], a, v)
    movel(p[x_c + 0.063050, y_c + -0.089671, z_c, rx, ry, rz], a, v)
    movel(p[x_c + 0.063447, y_c + -0.090123, z_c, rx, ry, rz], a, v)
    movel(p[x_c + 0.063866, y_c + -0.090581, z_c, rx, ry, rz], a, v)
    movel(p[x_c + 0.064306, y_c + -0.091047, z_c, rx, ry, rz], a, v)
    movel(p[x_c + 0.064769, y_c + -0.091523, z_c, rx, ry, rz], a, v)
    movel(p[x_c + 0.065255, y_c + -0.092009, z_c, rx, ry, rz], a, v)
    movel(p[x_c + 0.065765, y_c + -0.092506, z_c, rx, ry, rz], a, v)
    movel(p[x_c + 0.066298, y_c + -0.093015, z_c, rx, ry, rz], a, v)
    movel(p[x_c + 0.066856, y_c + -0.093537, z_c, rx, ry, rz], a, v)
    movel(p[x_c + 0.067438, y_c + -0.094074, z_c, rx, ry, rz], a, v)
    movel(p[x_c + 0.068047, y_c + -0.094626, z_c, rx, ry, rz], a, v)
    movel(p[x_c + 0.068681, y_c + -0.095194, z_c, rx, ry, rz], a, v)
    movel(p[x_c + 0.069341, y_c + -0.095779, z_c, rx, ry, rz], a, v)
    movel(p[x_c + 0.070028, y_c + -0.096383, z_c, rx, ry, rz], a, v)
    movel(p[x_c + 0.070743, y_c + -0.097006, z_c, rx, ry, rz], a, v)
    movel(p[x_c + 0.071485, y_c + -0.097649, z_c, rx, ry, rz], a, v)
    movel(p[x_c + 0.071485, y_c + -0.097649, z_c, rx, ry, rz], a, v)
    movel(p[x_c + 0.071659, y_c + -0.097799, z_c, rx, ry, rz], a, v)
    movel(p[x_c + 0.071842, y_c + -0.097958, z_c, rx, ry, rz], a, v)
    movel(p[x_c + 0.072034, y_c + -0.098124, z_c, rx, ry, rz], a, v)
    movel(p[x_c + 0.072234, y_c + -0.098298, z_c, rx, ry, rz], a, v)
    movel(p[x_c + 0.072443, y_c + -0.098479, z_c, rx, ry, rz], a, v)
    movel(p[x_c + 0.072660, y_c + -0.098667, z_c, rx, ry, rz], a, v)
    movel(p[x_c + 0.072885, y_c + -0.098862, z_c, rx, ry, rz], a, v)
    movel(p[x_c + 0.073116, y_c + -0.099064, z_c, rx, ry, rz], a, v)
    movel(p[x_c + 0.073355, y_c + -0.099271, z_c, rx, ry, rz], a, v)
    movel(p[x_c + 0.073600, y_c + -0.099484, z_c, rx, ry, rz], a, v)
    movel(p[x_c + 0.073851, y_c + -0.099703, z_c, rx, ry, rz], a, v)
    movel(p[x_c + 0.074108, y_c + -0.099927, z_c, rx, ry, rz], a, v)
    movel(p[x_c + 0.074370, y_c + -0.100155, z_c, rx, ry, rz], a, v)
    movel(p[x_c + 0.074637, y_c + -0.100388, z_c, rx, ry, rz], a, v)
    movel(p[x_c + 0.074910, y_c + -0.100625, z_c, rx, ry, rz], a, v)
    movel(p[x_c + 0.075186, y_c + -0.100867, z_c, rx, ry, rz], a, v)
    movel(p[x_c + 0.075467, y_c + -0.101111, z_c, rx, ry, rz], a, v)
    movel(p[x_c + 0.075751, y_c + -0.101359, z_c, rx, ry, rz], a, v)
    movel(p[x_c + 0.076038, y_c + -0.101610, z_c, rx, ry, rz], a, v)
    movel(p[x_c + 0.076329, y_c + -0.101864, z_c, rx, ry, rz], a, v)
    movel(p[x_c + 0.076622, y_c + -0.102119, z_c, rx, ry, rz], a, v)
    movel(p[x_c + 0.076917, y_c + -0.102377, z_c, rx, ry, rz], a, v)
    movel(p[x_c + 0.077214, y_c + -0.102637, z_c, rx, ry, rz], a, v)
    movel(p[x_c + 0.077512, y_c + -0.102898, z_c, rx, ry, rz], a, v)
    movel(p[x_c + 0.077812, y_c + -0.103160, z_c, rx, ry, rz], a, v)
    movel(p[x_c + 0.078112, y_c + -0.103423, z_c, rx, ry, rz], a, v)
    movel(p[x_c + 0.078413, y_c + -0.103686, z_c, rx, ry, rz], a, v)
    movel(p[x_c + 0.078714, y_c + -0.103949, z_c, rx, ry, rz], a, v)
    movel(p[x_c + 0.079015, y_c + -0.104212, z_c, rx, ry, rz], a, v)
    movel(p[x_c + 0.079315, y_c + -0.104475, z_c, rx, ry, rz], a, v)
    movel(p[x_c + 0.079614, y_c + -0.104737, z_c, rx, ry, rz], a, v)
    movel(p[x_c + 0.079912, y_c + -0.104998, z_c, rx, ry, rz], a, v)
    movel(p[x_c + 0.080208, y_c + -0.105257, z_c, rx, ry, rz], a, v)
    movel(p[x_c + 0.080501, y_c + -0.105515, z_c, rx, ry, rz], a, v)
    movel(p[x_c + 0.080793, y_c + -0.105770, z_c, rx, ry, rz], a, v)
    movel(p[x_c + 0.081082, y_c + -0.106023, z_c, rx, ry, rz], a, v)
    movel(p[x_c + 0.081367, y_c + -0.106274, z_c, rx, ry, rz], a, v)
    movel(p[x_c + 0.081649, y_c + -0.106521, z_c, rx, ry, rz], a, v)
    movel(p[x_c + 0.081927, y_c + -0.106766, z_c, rx, ry, rz], a, v)
    movel(p[x_c + 0.082201, y_c + -0.107006, z_c, rx, ry, rz], a, v)
    movel(p[x_c + 0.082471, y_c + -0.107243, z_c, rx, ry, rz], a, v)
    movel(p[x_c + 0.082735, y_c + -0.107475, z_c, rx, ry, rz], a, v)
    movel(p[x_c + 0.082995, y_c + -0.107703, z_c, rx, ry, rz], a, v)
    movel(p[x_c + 0.083248, y_c + -0.107926, z_c, rx, ry, rz], a, v)
    movel(p[x_c + 0.083496, y_c + -0.108144, z_c, rx, ry, rz], a, v)
    movel(p[x_c + 0.083737, y_c + -0.108356, z_c, rx, ry, rz], a, v)
    movel(p[x_c + 0.083971, y_c + -0.108563, z_c, rx, ry, rz], a, v)
    movel(p[x_c + 0.084199, y_c + -0.108764, z_c, rx, ry, rz], a, v)
    movel(p[x_c + 0.084419, y_c + -0.108958, z_c, rx, ry, rz], a, v)
    movel(p[x_c + 0.084419, y_c + -0.108958, z_c, rx, ry, rz], a, v)
    movel(p[x_c + 0.085000, y_c + -0.109470, z_c, rx, ry, rz], a, v)
    movel(p[x_c + 0.085000, y_c + -0.109470, z_c, rx, ry, rz], a, v)
    movel(p[x_c + 0.084330, y_c + -0.109136, z_c, rx, ry, rz], a, v)
    movel(p[x_c + 0.084330, y_c + -0.109136, z_c, rx, ry, rz], a, v)
    movel(p[x_c + 0.084305, y_c + -0.109123, z_c, rx, ry, rz], a, v)
    movel(p[x_c + 0.084275, y_c + -0.109107, z_c, rx, ry, rz], a, v)
    movel(p[x_c + 0.084241, y_c + -0.109088, z_c, rx, ry, rz], a, v)
    movel(p[x_c + 0.084202, y_c + -0.109066, z_c, rx, ry, rz], a, v)
    movel(p[x_c + 0.084158, y_c + -0.109040, z_c, rx, ry, rz], a, v)
    movel(p[x_c + 0.084110, y_c + -0.109012, z_c, rx, ry, rz], a, v)
    movel(p[x_c + 0.084057, y_c + -0.108981, z_c, rx, ry, rz], a, v)
    movel(p[x_c + 0.084001, y_c + -0.108947, z_c, rx, ry, rz], a, v)
    movel(p[x_c + 0.083940, y_c + -0.108910, z_c, rx, ry, rz], a, v)
    movel(p[x_c + 0.083875, y_c + -0.108871, z_c, rx, ry, rz], a, v)
    movel(p[x_c + 0.083806, y_c + -0.108829, z_c, rx, ry, rz], a, v)
    movel(p[x_c + 0.083733, y_c + -0.108784, z_c, rx, ry, rz], a, v)
    movel(p[x_c + 0.083656, y_c + -0.108736, z_c, rx, ry, rz], a, v)
    movel(p[x_c + 0.083576, y_c + -0.108687, z_c, rx, ry, rz], a, v)
    movel(p[x_c + 0.083492, y_c + -0.108634, z_c, rx, ry, rz], a, v)
    movel(p[x_c + 0.083405, y_c + -0.108580, z_c, rx, ry, rz], a, v)
    movel(p[x_c + 0.083314, y_c + -0.108523, z_c, rx, ry, rz], a, v)
    movel(p[x_c + 0.083219, y_c + -0.108464, z_c, rx, ry, rz], a, v)
    movel(p[x_c + 0.083122, y_c + -0.108402, z_c, rx, ry, rz], a, v)
    movel(p[x_c + 0.083021, y_c + -0.108339, z_c, rx, ry, rz], a, v)
    movel(p[x_c + 0.082918, y_c + -0.108273, z_c, rx, ry, rz], a, v)
    movel(p[x_c + 0.082811, y_c + -0.108206, z_c, rx, ry, rz], a, v)
    movel(p[x_c + 0.082702, y_c + -0.108136, z_c, rx, ry, rz], a, v)
    movel(p[x_c + 0.082589, y_c + -0.108065, z_c, rx, ry, rz], a, v)
    movel(p[x_c + 0.082474, y_c + -0.107991, z_c, rx, ry, rz], a, v)
    movel(p[x_c + 0.082357, y_c + -0.107916, z_c, rx, ry, rz], a, v)
    movel(p[x_c + 0.082237, y_c + -0.107839, z_c, rx, ry, rz], a, v)
    movel(p[x_c + 0.082114, y_c + -0.107761, z_c, rx, ry, rz], a, v)
    movel(p[x_c + 0.081990, y_c + -0.107681, z_c, rx, ry, rz], a, v)
    movel(p[x_c + 0.081863, y_c + -0.107599, z_c, rx, ry, rz], a, v)
    movel(p[x_c + 0.081734, y_c + -0.107516, z_c, rx, ry, rz], a, v)
    movel(p[x_c + 0.081602, y_c + -0.107432, z_c, rx, ry, rz], a, v)
    movel(p[x_c + 0.081469, y_c + -0.107346, z_c, rx, ry, rz], a, v)
    movel(p[x_c + 0.081334, y_c + -0.107259, z_c, rx, ry, rz], a, v)
    movel(p[x_c + 0.081198, y_c + -0.107170, z_c, rx, ry, rz], a, v)
    movel(p[x_c + 0.081059, y_c + -0.107080, z_c, rx, ry, rz], a, v)
    movel(p[x_c + 0.080919, y_c + -0.106990, z_c, rx, ry, rz], a, v)
    movel(p[x_c + 0.080778, y_c + -0.106898, z_c, rx, ry, rz], a, v)
    movel(p[x_c + 0.080635, y_c + -0.106805, z_c, rx, ry, rz], a, v)
    movel(p[x_c + 0.080491, y_c + -0.106711, z_c, rx, ry, rz], a, v)
    movel(p[x_c + 0.080346, y_c + -0.106616, z_c, rx, ry, rz], a, v)
    movel(p[x_c + 0.080199, y_c + -0.106521, z_c, rx, ry, rz], a, v)
    movel(p[x_c + 0.080052, y_c + -0.106425, z_c, rx, ry, rz], a, v)
    movel(p[x_c + 0.079904, y_c + -0.106327, z_c, rx, ry, rz], a, v)
    movel(p[x_c + 0.079754, y_c + -0.106230, z_c, rx, ry, rz], a, v)
    movel(p[x_c + 0.079604, y_c + -0.106131, z_c, rx, ry, rz], a, v)
    movel(p[x_c + 0.079454, y_c + -0.106033, z_c, rx, ry, rz], a, v)
    movel(p[x_c + 0.079303, y_c + -0.105933, z_c, rx, ry, rz], a, v)
    movel(p[x_c + 0.079151, y_c + -0.105833, z_c, rx, ry, rz], a, v)
    movel(p[x_c + 0.079151, y_c + -0.105833, z_c, rx, ry, rz], a, v)
    movel(p[x_c + 0.078888, y_c + -0.105660, z_c, rx, ry, rz], a, v)
    movel(p[x_c + 0.078630, y_c + -0.105491, z_c, rx, ry, rz], a, v)
    movel(p[x_c + 0.078378, y_c + -0.105325, z_c, rx, ry, rz], a, v)
    movel(p[x_c + 0.078132, y_c + -0.105163, z_c, rx, ry, rz], a, v)
    movel(p[x_c + 0.077891, y_c + -0.105005, z_c, rx, ry, rz], a, v)
    movel(p[x_c + 0.077655, y_c + -0.104850, z_c, rx, ry, rz], a, v)
    movel(p[x_c + 0.077425, y_c + -0.104699, z_c, rx, ry, rz], a, v)
    movel(p[x_c + 0.077200, y_c + -0.104552, z_c, rx, ry, rz], a, v)
    movel(p[x_c + 0.076981, y_c + -0.104408, z_c, rx, ry, rz], a, v)
    movel(p[x_c + 0.076767, y_c + -0.104268, z_c, rx, ry, rz], a, v)
    movel(p[x_c + 0.076558, y_c + -0.104132, z_c, rx, ry, rz], a, v)
    movel(p[x_c + 0.076355, y_c + -0.103999, z_c, rx, ry, rz], a, v)
    movel(p[x_c + 0.076156, y_c + -0.103869, z_c, rx, ry, rz], a, v)
    movel(p[x_c + 0.075963, y_c + -0.103744, z_c, rx, ry, rz], a, v)
    movel(p[x_c + 0.075776, y_c + -0.103621, z_c, rx, ry, rz], a, v)
    movel(p[x_c + 0.075593, y_c + -0.103502, z_c, rx, ry, rz], a, v)
    movel(p[x_c + 0.075416, y_c + -0.103387, z_c, rx, ry, rz], a, v)
    movel(p[x_c + 0.075244, y_c + -0.103275, z_c, rx, ry, rz], a, v)
    movel(p[x_c + 0.075077, y_c + -0.103167, z_c, rx, ry, rz], a, v)
    movel(p[x_c + 0.074915, y_c + -0.103062, z_c, rx, ry, rz], a, v)
    movel(p[x_c + 0.074758, y_c + -0.102961, z_c, rx, ry, rz], a, v)
    movel(p[x_c + 0.074606, y_c + -0.102863, z_c, rx, ry, rz], a, v)
    movel(p[x_c + 0.074459, y_c + -0.102768, z_c, rx, ry, rz], a, v)
    movel(p[x_c + 0.074317, y_c + -0.102677, z_c, rx, ry, rz], a, v)
    movel(p[x_c + 0.074180, y_c + -0.102589, z_c, rx, ry, rz], a, v)
    movel(p[x_c + 0.074048, y_c + -0.102504, z_c, rx, ry, rz], a, v)
    movel(p[x_c + 0.073921, y_c + -0.102423, z_c, rx, ry, rz], a, v)
    movel(p[x_c + 0.073799, y_c + -0.102345, z_c, rx, ry, rz], a, v)
    movel(p[x_c + 0.073682, y_c + -0.102271, z_c, rx, ry, rz], a, v)
    movel(p[x_c + 0.073570, y_c + -0.102200, z_c, rx, ry, rz], a, v)
    movel(p[x_c + 0.073462, y_c + -0.102132, z_c, rx, ry, rz], a, v)
    movel(p[x_c + 0.073359, y_c + -0.102067, z_c, rx, ry, rz], a, v)
    movel(p[x_c + 0.073261, y_c + -0.102005, z_c, rx, ry, rz], a, v)
    movel(p[x_c + 0.073168, y_c + -0.101947, z_c, rx, ry, rz], a, v)
    movel(p[x_c + 0.073079, y_c + -0.101892, z_c, rx, ry, rz], a, v)
    movel(p[x_c + 0.072996, y_c + -0.101840, z_c, rx, ry, rz], a, v)
    movel(p[x_c + 0.072916, y_c + -0.101792, z_c, rx, ry, rz], a, v)
    movel(p[x_c + 0.072842, y_c + -0.101746, z_c, rx, ry, rz], a, v)
    movel(p[x_c + 0.072772, y_c + -0.101704, z_c, rx, ry, rz], a, v)
    movel(p[x_c + 0.072707, y_c + -0.101664, z_c, rx, ry, rz], a, v)
    movel(p[x_c + 0.072646, y_c + -0.101628, z_c, rx, ry, rz], a, v)
    movel(p[x_c + 0.072590, y_c + -0.101595, z_c, rx, ry, rz], a, v)
    movel(p[x_c + 0.072538, y_c + -0.101565, z_c, rx, ry, rz], a, v)
    movel(p[x_c + 0.072491, y_c + -0.101539, z_c, rx, ry, rz], a, v)
    movel(p[x_c + 0.072448, y_c + -0.101515, z_c, rx, ry, rz], a, v)
    movel(p[x_c + 0.072410, y_c + -0.101494, z_c, rx, ry, rz], a, v)
    movel(p[x_c + 0.072376, y_c + -0.101476, z_c, rx, ry, rz], a, v)
    movel(p[x_c + 0.072347, y_c + -0.101461, z_c, rx, ry, rz], a, v)
    movel(p[x_c + 0.072322, y_c + -0.101450, z_c, rx, ry, rz], a, v)
    movel(p[x_c + 0.072322, y_c + -0.101450, z_c, rx, ry, rz], a, v)
    movel(p[x_c + 0.072319, y_c + -0.101450, z_c, rx, ry, rz], a, v)
    movel(p[x_c + 0.072322, y_c + -0.101456, z_c, rx, ry, rz], a, v)
    movel(p[x_c + 0.072332, y_c + -0.101468, z_c, rx, ry, rz], a, v)
    movel(p[x_c + 0.072347, y_c + -0.101487, z_c, rx, ry, rz], a, v)
    movel(p[x_c + 0.072368, y_c + -0.101510, z_c, rx, ry, rz], a, v)
    movel(p[x_c + 0.072395, y_c + -0.101540, z_c, rx, ry, rz], a, v)
    movel(p[x_c + 0.072427, y_c + -0.101575, z_c, rx, ry, rz], a, v)
    movel(p[x_c + 0.072465, y_c + -0.101615, z_c, rx, ry, rz], a, v)
    movel(p[x_c + 0.072508, y_c + -0.101661, z_c, rx, ry, rz], a, v)
    movel(p[x_c + 0.072557, y_c + -0.101712, z_c, rx, ry, rz], a, v)
    movel(p[x_c + 0.072611, y_c + -0.101768, z_c, rx, ry, rz], a, v)
    movel(p[x_c + 0.072670, y_c + -0.101829, z_c, rx, ry, rz], a, v)
    movel(p[x_c + 0.072734, y_c + -0.101896, z_c, rx, ry, rz], a, v)
    movel(p[x_c + 0.072804, y_c + -0.101967, z_c, rx, ry, rz], a, v)
    movel(p[x_c + 0.072878, y_c + -0.102043, z_c, rx, ry, rz], a, v)
    movel(p[x_c + 0.072957, y_c + -0.102123, z_c, rx, ry, rz], a, v)
    movel(p[x_c + 0.073040, y_c + -0.102208, z_c, rx, ry, rz], a, v)
    movel(p[x_c + 0.073128, y_c + -0.102298, z_c, rx, ry, rz], a, v)
    movel(p[x_c + 0.073221, y_c + -0.102392, z_c, rx, ry, rz], a, v)
    movel(p[x_c + 0.073318, y_c + -0.102490, z_c, rx, ry, rz], a, v)
    movel(p[x_c + 0.073419, y_c + -0.102593, z_c, rx, ry, rz], a, v)
    movel(p[x_c + 0.073525, y_c + -0.102699, z_c, rx, ry, rz], a, v)
    movel(p[x_c + 0.073635, y_c + -0.102810, z_c, rx, ry, rz], a, v)
    movel(p[x_c + 0.073748, y_c + -0.102925, z_c, rx, ry, rz], a, v)
    movel(p[x_c + 0.073866, y_c + -0.103043, z_c, rx, ry, rz], a, v)
    movel(p[x_c + 0.073987, y_c + -0.103165, z_c, rx, ry, rz], a, v)
    movel(p[x_c + 0.074113, y_c + -0.103291, z_c, rx, ry, rz], a, v)
    movel(p[x_c + 0.074242, y_c + -0.103420, z_c, rx, ry, rz], a, v)
    movel(p[x_c + 0.074374, y_c + -0.103553, z_c, rx, ry, rz], a, v)
    movel(p[x_c + 0.074510, y_c + -0.103689, z_c, rx, ry, rz], a, v)
    movel(p[x_c + 0.074649, y_c + -0.103828, z_c, rx, ry, rz], a, v)
    movel(p[x_c + 0.074792, y_c + -0.103971, z_c, rx, ry, rz], a, v)
    movel(p[x_c + 0.074938, y_c + -0.104116, z_c, rx, ry, rz], a, v)
    movel(p[x_c + 0.075086, y_c + -0.104265, z_c, rx, ry, rz], a, v)
    movel(p[x_c + 0.075238, y_c + -0.104416, z_c, rx, ry, rz], a, v)
    movel(p[x_c + 0.075393, y_c + -0.104571, z_c, rx, ry, rz], a, v)
    movel(p[x_c + 0.075550, y_c + -0.104727, z_c, rx, ry, rz], a, v)
    movel(p[x_c + 0.075711, y_c + -0.104887, z_c, rx, ry, rz], a, v)
    movel(p[x_c + 0.075873, y_c + -0.105049, z_c, rx, ry, rz], a, v)
    movel(p[x_c + 0.076039, y_c + -0.105213, z_c, rx, ry, rz], a, v)
    movel(p[x_c + 0.076206, y_c + -0.105380, z_c, rx, ry, rz], a, v)
    movel(p[x_c + 0.076376, y_c + -0.105548, z_c, rx, ry, rz], a, v)
    movel(p[x_c + 0.076549, y_c + -0.105719, z_c, rx, ry, rz], a, v)
    movel(p[x_c + 0.076723, y_c + -0.105892, z_c, rx, ry, rz], a, v)
    movel(p[x_c + 0.076900, y_c + -0.106067, z_c, rx, ry, rz], a, v)
    movel(p[x_c + 0.077078, y_c + -0.106244, z_c, rx, ry, rz], a, v)
    movel(p[x_c + 0.077258, y_c + -0.106422, z_c, rx, ry, rz], a, v)
    movel(p[x_c + 0.077440, y_c + -0.106602, z_c, rx, ry, rz], a, v)
    movel(p[x_c + 0.077624, y_c + -0.106784, z_c, rx, ry, rz], a, v)
    movel(p[x_c + 0.077624, y_c + -0.106784, z_c, rx, ry, rz], a, v)
    movel(p[x_c + 0.077808, y_c + -0.106966, z_c, rx, ry, rz], a, v)
    movel(p[x_c + 0.077990, y_c + -0.107147, z_c, rx, ry, rz], a, v)
    movel(p[x_c + 0.078171, y_c + -0.107326, z_c, rx, ry, rz], a, v)
    movel(p[x_c + 0.078350, y_c + -0.107505, z_c, rx, ry, rz], a, v)
    movel(p[x_c + 0.078527, y_c + -0.107682, z_c, rx, ry, rz], a, v)
    movel(p[x_c + 0.078703, y_c + -0.107858, z_c, rx, ry, rz], a, v)
    movel(p[x_c + 0.078876, y_c + -0.108032, z_c, rx, ry, rz], a, v)
    movel(p[x_c + 0.079048, y_c + -0.108204, z_c, rx, ry, rz], a, v)
    movel(p[x_c + 0.079217, y_c + -0.108375, z_c, rx, ry, rz], a, v)
    movel(p[x_c + 0.079384, y_c + -0.108544, z_c, rx, ry, rz], a, v)
    movel(p[x_c + 0.079549, y_c + -0.108711, z_c, rx, ry, rz], a, v)
    movel(p[x_c + 0.079711, y_c + -0.108876, z_c, rx, ry, rz], a, v)
    movel(p[x_c + 0.079871, y_c + -0.109038, z_c, rx, ry, rz], a, v)
    movel(p[x_c + 0.080028, y_c + -0.109199, z_c, rx, ry, rz], a, v)
    movel(p[x_c + 0.080182, y_c + -0.109357, z_c, rx, ry, rz], a, v)
    movel(p[x_c + 0.080334, y_c + -0.109513, z_c, rx, ry, rz], a, v)
    movel(p[x_c + 0.080482, y_c + -0.109666, z_c, rx, ry, rz], a, v)
    movel(p[x_c + 0.080628, y_c + -0.109816, z_c, rx, ry, rz], a, v)
    movel(p[x_c + 0.080770, y_c + -0.109964, z_c, rx, ry, rz], a, v)
    movel(p[x_c + 0.080909, y_c + -0.110108, z_c, rx, ry, rz], a, v)
    movel(p[x_c + 0.081045, y_c + -0.110250, z_c, rx, ry, rz], a, v)
    movel(p[x_c + 0.081178, y_c + -0.110389, z_c, rx, ry, rz], a, v)
    movel(p[x_c + 0.081307, y_c + -0.110524, z_c, rx, ry, rz], a, v)
    movel(p[x_c + 0.081432, y_c + -0.110656, z_c, rx, ry, rz], a, v)
    movel(p[x_c + 0.081553, y_c + -0.110785, z_c, rx, ry, rz], a, v)
    movel(p[x_c + 0.081671, y_c + -0.110910, z_c, rx, ry, rz], a, v)
    movel(p[x_c + 0.081785, y_c + -0.111031, z_c, rx, ry, rz], a, v)
    movel(p[x_c + 0.081895, y_c + -0.111149, z_c, rx, ry, rz], a, v)
    movel(p[x_c + 0.082001, y_c + -0.111263, z_c, rx, ry, rz], a, v)
    movel(p[x_c + 0.082102, y_c + -0.111374, z_c, rx, ry, rz], a, v)
    movel(p[x_c + 0.082199, y_c + -0.111480, z_c, rx, ry, rz], a, v)
    movel(p[x_c + 0.082292, y_c + -0.111582, z_c, rx, ry, rz], a, v)
    movel(p[x_c + 0.082380, y_c + -0.111679, z_c, rx, ry, rz], a, v)
    movel(p[x_c + 0.082464, y_c + -0.111773, z_c, rx, ry, rz], a, v)
    movel(p[x_c + 0.082543, y_c + -0.111862, z_c, rx, ry, rz], a, v)
    movel(p[x_c + 0.082617, y_c + -0.111946, z_c, rx, ry, rz], a, v)
    movel(p[x_c + 0.082687, y_c + -0.112026, z_c, rx, ry, rz], a, v)
    movel(p[x_c + 0.082751, y_c + -0.112101, z_c, rx, ry, rz], a, v)
    movel(p[x_c + 0.082810, y_c + -0.112171, z_c, rx, ry, rz], a, v)
    movel(p[x_c + 0.082864, y_c + -0.112236, z_c, rx, ry, rz], a, v)
    movel(p[x_c + 0.082913, y_c + -0.112296, z_c, rx, ry, rz], a, v)
    movel(p[x_c + 0.082957, y_c + -0.112351, z_c, rx, ry, rz], a, v)
    movel(p[x_c + 0.082995, y_c + -0.112401, z_c, rx, ry, rz], a, v)
    movel(p[x_c + 0.083027, y_c + -0.112445, z_c, rx, ry, rz], a, v)
    movel(p[x_c + 0.083054, y_c + -0.112484, z_c, rx, ry, rz], a, v)
    movel(p[x_c + 0.083075, y_c + -0.112517, z_c, rx, ry, rz], a, v)
    movel(p[x_c + 0.083090, y_c + -0.112545, z_c, rx, ry, rz], a, v)
    movel(p[x_c + 0.083099, y_c + -0.112567, z_c, rx, ry, rz], a, v)
    movel(p[x_c + 0.083102, y_c + -0.112583, z_c, rx, ry, rz], a, v)
    movel(p[x_c + 0.083102, y_c + -0.112583, z_c, rx, ry, rz], a, v)
    movel(p[x_c + 0.083102, y_c + -0.112596, z_c, rx, ry, rz], a, v)
    movel(p[x_c + 0.083101, y_c + -0.112609, z_c, rx, ry, rz], a, v)
    movel(p[x_c + 0.083100, y_c + -0.112622, z_c, rx, ry, rz], a, v)
    movel(p[x_c + 0.083099, y_c + -0.112636, z_c, rx, ry, rz], a, v)
    movel(p[x_c + 0.083097, y_c + -0.112650, z_c, rx, ry, rz], a, v)
    movel(p[x_c + 0.083095, y_c + -0.112664, z_c, rx, ry, rz], a, v)
    movel(p[x_c + 0.083093, y_c + -0.112678, z_c, rx, ry, rz], a, v)
    movel(p[x_c + 0.083090, y_c + -0.112692, z_c, rx, ry, rz], a, v)
    movel(p[x_c + 0.083087, y_c + -0.112707, z_c, rx, ry, rz], a, v)
    movel(p[x_c + 0.083084, y_c + -0.112721, z_c, rx, ry, rz], a, v)
    movel(p[x_c + 0.083080, y_c + -0.112736, z_c, rx, ry, rz], a, v)
    movel(p[x_c + 0.083076, y_c + -0.112750, z_c, rx, ry, rz], a, v)
    movel(p[x_c + 0.083072, y_c + -0.112765, z_c, rx, ry, rz], a, v)
    movel(p[x_c + 0.083067, y_c + -0.112780, z_c, rx, ry, rz], a, v)
    movel(p[x_c + 0.083062, y_c + -0.112795, z_c, rx, ry, rz], a, v)
    movel(p[x_c + 0.083057, y_c + -0.112810, z_c, rx, ry, rz], a, v)
    movel(p[x_c + 0.083052, y_c + -0.112825, z_c, rx, ry, rz], a, v)
    movel(p[x_c + 0.083046, y_c + -0.112840, z_c, rx, ry, rz], a, v)
    movel(p[x_c + 0.083040, y_c + -0.112855, z_c, rx, ry, rz], a, v)
    movel(p[x_c + 0.083034, y_c + -0.112870, z_c, rx, ry, rz], a, v)
    movel(p[x_c + 0.083027, y_c + -0.112885, z_c, rx, ry, rz], a, v)
    movel(p[x_c + 0.083020, y_c + -0.112900, z_c, rx, ry, rz], a, v)
    movel(p[x_c + 0.083013, y_c + -0.112915, z_c, rx, ry, rz], a, v)
    movel(p[x_c + 0.083006, y_c + -0.112930, z_c, rx, ry, rz], a, v)
    movel(p[x_c + 0.082998, y_c + -0.112944, z_c, rx, ry, rz], a, v)
    movel(p[x_c + 0.082990, y_c + -0.112959, z_c, rx, ry, rz], a, v)
    movel(p[x_c + 0.082982, y_c + -0.112974, z_c, rx, ry, rz], a, v)
    movel(p[x_c + 0.082974, y_c + -0.112988, z_c, rx, ry, rz], a, v)
    movel(p[x_c + 0.082966, y_c + -0.113003, z_c, rx, ry, rz], a, v)
    movel(p[x_c + 0.082957, y_c + -0.113017, z_c, rx, ry, rz], a, v)
    movel(p[x_c + 0.082948, y_c + -0.113031, z_c, rx, ry, rz], a, v)
    movel(p[x_c + 0.082939, y_c + -0.113045, z_c, rx, ry, rz], a, v)
    movel(p[x_c + 0.082930, y_c + -0.113059, z_c, rx, ry, rz], a, v)
    movel(p[x_c + 0.082920, y_c + -0.113073, z_c, rx, ry, rz], a, v)
    movel(p[x_c + 0.082911, y_c + -0.113086, z_c, rx, ry, rz], a, v)
    movel(p[x_c + 0.082901, y_c + -0.113100, z_c, rx, ry, rz], a, v)
    movel(p[x_c + 0.082891, y_c + -0.113113, z_c, rx, ry, rz], a, v)
    movel(p[x_c + 0.082881, y_c + -0.113126, z_c, rx, ry, rz], a, v)
    movel(p[x_c + 0.082871, y_c + -0.113138, z_c, rx, ry, rz], a, v)
    movel(p[x_c + 0.082860, y_c + -0.113151, z_c, rx, ry, rz], a, v)
    movel(p[x_c + 0.082850, y_c + -0.113163, z_c, rx, ry, rz], a, v)
    movel(p[x_c + 0.082839, y_c + -0.113175, z_c, rx, ry, rz], a, v)
    movel(p[x_c + 0.082828, y_c + -0.113186, z_c, rx, ry, rz], a, v)
    movel(p[x_c + 0.082817, y_c + -0.113198, z_c, rx, ry, rz], a, v)
    movel(p[x_c + 0.082806, y_c + -0.113209, z_c, rx, ry, rz], a, v)
    movel(p[x_c + 0.082795, y_c + -0.113220, z_c, rx, ry, rz], a, v)
    movel(p[x_c + 0.082784, y_c + -0.113230, z_c, rx, ry, rz], a, v)
    movel(p[x_c + 0.082772, y_c + -0.113240, z_c, rx, ry, rz], a, v)
    movel(p[x_c + 0.082761, y_c + -0.113250, z_c, rx, ry, rz], a, v)
    movel(p[x_c + 0.082761, y_c + -0.113250, z_c, rx, ry, rz], a, v)
    movel(p[x_c + 0.082744, y_c + -0.113264, z_c, rx, ry, rz], a, v)
    movel(p[x_c + 0.082727, y_c + -0.113277, z_c, rx, ry, rz], a, v)
    movel(p[x_c + 0.082711, y_c + -0.113290, z_c, rx, ry, rz], a, v)
    movel(p[x_c + 0.082695, y_c + -0.113302, z_c, rx, ry, rz], a, v)
    movel(p[x_c + 0.082679, y_c + -0.113313, z_c, rx, ry, rz], a, v)
    movel(p[x_c + 0.082663, y_c + -0.113324, z_c, rx, ry, rz], a, v)
    movel(p[x_c + 0.082647, y_c + -0.113334, z_c, rx, ry, rz], a, v)
    movel(p[x_c + 0.082632, y_c + -0.113343, z_c, rx, ry, rz], a, v)
    movel(p[x_c + 0.082617, y_c + -0.113351, z_c, rx, ry, rz], a, v)
    movel(p[x_c + 0.082602, y_c + -0.113359, z_c, rx, ry, rz], a, v)
    movel(p[x_c + 0.082587, y_c + -0.113367, z_c, rx, ry, rz], a, v)
    movel(p[x_c + 0.082573, y_c + -0.113373, z_c, rx, ry, rz], a, v)
    movel(p[x_c + 0.082558, y_c + -0.113379, z_c, rx, ry, rz], a, v)
    movel(p[x_c + 0.082543, y_c + -0.113384, z_c, rx, ry, rz], a, v)
    movel(p[x_c + 0.082529, y_c + -0.113388, z_c, rx, ry, rz], a, v)
    movel(p[x_c + 0.082514, y_c + -0.113392, z_c, rx, ry, rz], a, v)
    movel(p[x_c + 0.082500, y_c + -0.113395, z_c, rx, ry, rz], a, v)
    movel(p[x_c + 0.082486, y_c + -0.113397, z_c, rx, ry, rz], a, v)
    movel(p[x_c + 0.082471, y_c + -0.113399, z_c, rx, ry, rz], a, v)
    movel(p[x_c + 0.082457, y_c + -0.113399, z_c, rx, ry, rz], a, v)
    movel(p[x_c + 0.082442, y_c + -0.113399, z_c, rx, ry, rz], a, v)
    movel(p[x_c + 0.082427, y_c + -0.113399, z_c, rx, ry, rz], a, v)
    movel(p[x_c + 0.082413, y_c + -0.113397, z_c, rx, ry, rz], a, v)
    movel(p[x_c + 0.082398, y_c + -0.113395, z_c, rx, ry, rz], a, v)
    movel(p[x_c + 0.082383, y_c + -0.113392, z_c, rx, ry, rz], a, v)
    movel(p[x_c + 0.082367, y_c + -0.113388, z_c, rx, ry, rz], a, v)
    movel(p[x_c + 0.082352, y_c + -0.113384, z_c, rx, ry, rz], a, v)
    movel(p[x_c + 0.082336, y_c + -0.113379, z_c, rx, ry, rz], a, v)
    movel(p[x_c + 0.082320, y_c + -0.113373, z_c, rx, ry, rz], a, v)
    movel(p[x_c + 0.082304, y_c + -0.113366, z_c, rx, ry, rz], a, v)
    movel(p[x_c + 0.082288, y_c + -0.113358, z_c, rx, ry, rz], a, v)
    movel(p[x_c + 0.082271, y_c + -0.113350, z_c, rx, ry, rz], a, v)
    movel(p[x_c + 0.082254, y_c + -0.113341, z_c, rx, ry, rz], a, v)
    movel(p[x_c + 0.082237, y_c + -0.113331, z_c, rx, ry, rz], a, v)
    movel(p[x_c + 0.082219, y_c + -0.113320, z_c, rx, ry, rz], a, v)
    movel(p[x_c + 0.082201, y_c + -0.113309, z_c, rx, ry, rz], a, v)
    movel(p[x_c + 0.082183, y_c + -0.113297, z_c, rx, ry, rz], a, v)
    movel(p[x_c + 0.082164, y_c + -0.113283, z_c, rx, ry, rz], a, v)
    movel(p[x_c + 0.082145, y_c + -0.113270, z_c, rx, ry, rz], a, v)
    movel(p[x_c + 0.082125, y_c + -0.113255, z_c, rx, ry, rz], a, v)
    movel(p[x_c + 0.082105, y_c + -0.113239, z_c, rx, ry, rz], a, v)
    movel(p[x_c + 0.082084, y_c + -0.113223, z_c, rx, ry, rz], a, v)
    movel(p[x_c + 0.082063, y_c + -0.113206, z_c, rx, ry, rz], a, v)
    movel(p[x_c + 0.082041, y_c + -0.113188, z_c, rx, ry, rz], a, v)
    movel(p[x_c + 0.082019, y_c + -0.113169, z_c, rx, ry, rz], a, v)
    movel(p[x_c + 0.081996, y_c + -0.113149, z_c, rx, ry, rz], a, v)
    movel(p[x_c + 0.081973, y_c + -0.113129, z_c, rx, ry, rz], a, v)
    movel(p[x_c + 0.081949, y_c + -0.113107, z_c, rx, ry, rz], a, v)
    movel(p[x_c + 0.081924, y_c + -0.113085, z_c, rx, ry, rz], a, v)
    movel(p[x_c + 0.081924, y_c + -0.113085, z_c, rx, ry, rz], a, v)
    movel(p[x_c + 0.081905, y_c + -0.113069, z_c, rx, ry, rz], a, v)
    movel(p[x_c + 0.081882, y_c + -0.113049, z_c, rx, ry, rz], a, v)
    movel(p[x_c + 0.081855, y_c + -0.113027, z_c, rx, ry, rz], a, v)
    movel(p[x_c + 0.081824, y_c + -0.113002, z_c, rx, ry, rz], a, v)
    movel(p[x_c + 0.081789, y_c + -0.112974, z_c, rx, ry, rz], a, v)
    movel(p[x_c + 0.081750, y_c + -0.112944, z_c, rx, ry, rz], a, v)
    movel(p[x_c + 0.081707, y_c + -0.112911, z_c, rx, ry, rz], a, v)
    movel(p[x_c + 0.081660, y_c + -0.112876, z_c, rx, ry, rz], a, v)
    movel(p[x_c + 0.081610, y_c + -0.112838, z_c, rx, ry, rz], a, v)
    movel(p[x_c + 0.081556, y_c + -0.112798, z_c, rx, ry, rz], a, v)
    movel(p[x_c + 0.081499, y_c + -0.112755, z_c, rx, ry, rz], a, v)
    movel(p[x_c + 0.081439, y_c + -0.112710, z_c, rx, ry, rz], a, v)
    movel(p[x_c + 0.081375, y_c + -0.112663, z_c, rx, ry, rz], a, v)
    movel(p[x_c + 0.081308, y_c + -0.112614, z_c, rx, ry, rz], a, v)
    movel(p[x_c + 0.081237, y_c + -0.112562, z_c, rx, ry, rz], a, v)
    movel(p[x_c + 0.081164, y_c + -0.112509, z_c, rx, ry, rz], a, v)
    movel(p[x_c + 0.081087, y_c + -0.112453, z_c, rx, ry, rz], a, v)
    movel(p[x_c + 0.081008, y_c + -0.112396, z_c, rx, ry, rz], a, v)
    movel(p[x_c + 0.080926, y_c + -0.112336, z_c, rx, ry, rz], a, v)
    movel(p[x_c + 0.080841, y_c + -0.112275, z_c, rx, ry, rz], a, v)
    movel(p[x_c + 0.080753, y_c + -0.112212, z_c, rx, ry, rz], a, v)
    movel(p[x_c + 0.080663, y_c + -0.112147, z_c, rx, ry, rz], a, v)
    movel(p[x_c + 0.080570, y_c + -0.112080, z_c, rx, ry, rz], a, v)
    movel(p[x_c + 0.080475, y_c + -0.112012, z_c, rx, ry, rz], a, v)
    movel(p[x_c + 0.080377, y_c + -0.111943, z_c, rx, ry, rz], a, v)
    movel(p[x_c + 0.080277, y_c + -0.111871, z_c, rx, ry, rz], a, v)
    movel(p[x_c + 0.080175, y_c + -0.111799, z_c, rx, ry, rz], a, v)
    movel(p[x_c + 0.080070, y_c + -0.111725, z_c, rx, ry, rz], a, v)
    movel(p[x_c + 0.079964, y_c + -0.111649, z_c, rx, ry, rz], a, v)
    movel(p[x_c + 0.079855, y_c + -0.111573, z_c, rx, ry, rz], a, v)
    movel(p[x_c + 0.079745, y_c + -0.111495, z_c, rx, ry, rz], a, v)
    movel(p[x_c + 0.079633, y_c + -0.111416, z_c, rx, ry, rz], a, v)
    movel(p[x_c + 0.079519, y_c + -0.111335, z_c, rx, ry, rz], a, v)
    movel(p[x_c + 0.079403, y_c + -0.111254, z_c, rx, ry, rz], a, v)
    movel(p[x_c + 0.079286, y_c + -0.111172, z_c, rx, ry, rz], a, v)
    movel(p[x_c + 0.079167, y_c + -0.111088, z_c, rx, ry, rz], a, v)
    movel(p[x_c + 0.079047, y_c + -0.111004, z_c, rx, ry, rz], a, v)
    movel(p[x_c + 0.078926, y_c + -0.110919, z_c, rx, ry, rz], a, v)
    movel(p[x_c + 0.078803, y_c + -0.110833, z_c, rx, ry, rz], a, v)
    movel(p[x_c + 0.078679, y_c + -0.110747, z_c, rx, ry, rz], a, v)
    movel(p[x_c + 0.078554, y_c + -0.110660, z_c, rx, ry, rz], a, v)
    movel(p[x_c + 0.078427, y_c + -0.110572, z_c, rx, ry, rz], a, v)
    movel(p[x_c + 0.078300, y_c + -0.110484, z_c, rx, ry, rz], a, v)
    movel(p[x_c + 0.078172, y_c + -0.110395, z_c, rx, ry, rz], a, v)
    movel(p[x_c + 0.078043, y_c + -0.110305, z_c, rx, ry, rz], a, v)
    movel(p[x_c + 0.077914, y_c + -0.110216, z_c, rx, ry, rz], a, v)
    movel(p[x_c + 0.077784, y_c + -0.110126, z_c, rx, ry, rz], a, v)
    movel(p[x_c + 0.077653, y_c + -0.110035, z_c, rx, ry, rz], a, v)
    movel(p[x_c + 0.077522, y_c + -0.109945, z_c, rx, ry, rz], a, v)
    movel(p[x_c + 0.077522, y_c + -0.109945, z_c, rx, ry, rz], a, v)
    movel(p[x_c + 0.077390, y_c + -0.109854, z_c, rx, ry, rz], a, v)
    movel(p[x_c + 0.077258, y_c + -0.109763, z_c, rx, ry, rz], a, v)
    movel(p[x_c + 0.077127, y_c + -0.109672, z_c, rx, ry, rz], a, v)
    movel(p[x_c + 0.076995, y_c + -0.109582, z_c, rx, ry, rz], a, v)
    movel(p[x_c + 0.076864, y_c + -0.109491, z_c, rx, ry, rz], a, v)
    movel(p[x_c + 0.076733, y_c + -0.109400, z_c, rx, ry, rz], a, v)
    movel(p[x_c + 0.076602, y_c + -0.109310, z_c, rx, ry, rz], a, v)
    movel(p[x_c + 0.076472, y_c + -0.109220, z_c, rx, ry, rz], a, v)
    movel(p[x_c + 0.076342, y_c + -0.109131, z_c, rx, ry, rz], a, v)
    movel(p[x_c + 0.076213, y_c + -0.109041, z_c, rx, ry, rz], a, v)
    movel(p[x_c + 0.076085, y_c + -0.108953, z_c, rx, ry, rz], a, v)
    movel(p[x_c + 0.075957, y_c + -0.108865, z_c, rx, ry, rz], a, v)
    movel(p[x_c + 0.075830, y_c + -0.108777, z_c, rx, ry, rz], a, v)
    movel(p[x_c + 0.075705, y_c + -0.108690, z_c, rx, ry, rz], a, v)
    movel(p[x_c + 0.075580, y_c + -0.108604, z_c, rx, ry, rz], a, v)
    movel(p[x_c + 0.075457, y_c + -0.108518, z_c, rx, ry, rz], a, v)
    movel(p[x_c + 0.075335, y_c + -0.108434, z_c, rx, ry, rz], a, v)
    movel(p[x_c + 0.075214, y_c + -0.108350, z_c, rx, ry, rz], a, v)
    movel(p[x_c + 0.075094, y_c + -0.108268, z_c, rx, ry, rz], a, v)
    movel(p[x_c + 0.074977, y_c + -0.108186, z_c, rx, ry, rz], a, v)
    movel(p[x_c + 0.074860, y_c + -0.108105, z_c, rx, ry, rz], a, v)
    movel(p[x_c + 0.074746, y_c + -0.108026, z_c, rx, ry, rz], a, v)
    movel(p[x_c + 0.074633, y_c + -0.107948, z_c, rx, ry, rz], a, v)
    movel(p[x_c + 0.074522, y_c + -0.107871, z_c, rx, ry, rz], a, v)
    movel(p[x_c + 0.074413, y_c + -0.107795, z_c, rx, ry, rz], a, v)
    movel(p[x_c + 0.074306, y_c + -0.107721, z_c, rx, ry, rz], a, v)
    movel(p[x_c + 0.074201, y_c + -0.107648, z_c, rx, ry, rz], a, v)
    movel(p[x_c + 0.074099, y_c + -0.107577, z_c, rx, ry, rz], a, v)
    movel(p[x_c + 0.073998, y_c + -0.107507, z_c, rx, ry, rz], a, v)
    movel(p[x_c + 0.073900, y_c + -0.107439, z_c, rx, ry, rz], a, v)
    movel(p[x_c + 0.073805, y_c + -0.107373, z_c, rx, ry, rz], a, v)
    movel(p[x_c + 0.073712, y_c + -0.107308, z_c, rx, ry, rz], a, v)
    movel(p[x_c + 0.073622, y_c + -0.107245, z_c, rx, ry, rz], a, v)
    movel(p[x_c + 0.073534, y_c + -0.107184, z_c, rx, ry, rz], a, v)
    movel(p[x_c + 0.073450, y_c + -0.107125, z_c, rx, ry, rz], a, v)
    movel(p[x_c + 0.073368, y_c + -0.107068, z_c, rx, ry, rz], a, v)
    movel(p[x_c + 0.073289, y_c + -0.107013, z_c, rx, ry, rz], a, v)
    movel(p[x_c + 0.073214, y_c + -0.106960, z_c, rx, ry, rz], a, v)
    movel(p[x_c + 0.073141, y_c + -0.106910, z_c, rx, ry, rz], a, v)
    movel(p[x_c + 0.073072, y_c + -0.106861, z_c, rx, ry, rz], a, v)
    movel(p[x_c + 0.073006, y_c + -0.106815, z_c, rx, ry, rz], a, v)
    movel(p[x_c + 0.072944, y_c + -0.106771, z_c, rx, ry, rz], a, v)
    movel(p[x_c + 0.072885, y_c + -0.106730, z_c, rx, ry, rz], a, v)
    movel(p[x_c + 0.072829, y_c + -0.106691, z_c, rx, ry, rz], a, v)
    movel(p[x_c + 0.072778, y_c + -0.106655, z_c, rx, ry, rz], a, v)
    movel(p[x_c + 0.072730, y_c + -0.106621, z_c, rx, ry, rz], a, v)
    movel(p[x_c + 0.072686, y_c + -0.106590, z_c, rx, ry, rz], a, v)
    movel(p[x_c + 0.072646, y_c + -0.106562, z_c, rx, ry, rz], a, v)
    movel(p[x_c + 0.072610, y_c + -0.106537, z_c, rx, ry, rz], a, v)
    movel(p[x_c + 0.072610, y_c + -0.106537, z_c, rx, ry, rz], a, v)
    movel(p[x_c + 0.072554, y_c + -0.106497, z_c, rx, ry, rz], a, v)
    movel(p[x_c + 0.072501, y_c + -0.106459, z_c, rx, ry, rz], a, v)
    movel(p[x_c + 0.072450, y_c + -0.106422, z_c, rx, ry, rz], a, v)
    movel(p[x_c + 0.072401, y_c + -0.106388, z_c, rx, ry, rz], a, v)
    movel(p[x_c + 0.072354, y_c + -0.106355, z_c, rx, ry, rz], a, v)
    movel(p[x_c + 0.072310, y_c + -0.106324, z_c, rx, ry, rz], a, v)
    movel(p[x_c + 0.072269, y_c + -0.106295, z_c, rx, ry, rz], a, v)
    movel(p[x_c + 0.072230, y_c + -0.106268, z_c, rx, ry, rz], a, v)
    movel(p[x_c + 0.072193, y_c + -0.106242, z_c, rx, ry, rz], a, v)
    movel(p[x_c + 0.072159, y_c + -0.106219, z_c, rx, ry, rz], a, v)
    movel(p[x_c + 0.072127, y_c + -0.106197, z_c, rx, ry, rz], a, v)
    movel(p[x_c + 0.072098, y_c + -0.106178, z_c, rx, ry, rz], a, v)
    movel(p[x_c + 0.072071, y_c + -0.106160, z_c, rx, ry, rz], a, v)
    movel(p[x_c + 0.072047, y_c + -0.106144, z_c, rx, ry, rz], a, v)
    movel(p[x_c + 0.072025, y_c + -0.106130, z_c, rx, ry, rz], a, v)
    movel(p[x_c + 0.072006, y_c + -0.106119, z_c, rx, ry, rz], a, v)
    movel(p[x_c + 0.071989, y_c + -0.106109, z_c, rx, ry, rz], a, v)
    movel(p[x_c + 0.071975, y_c + -0.106101, z_c, rx, ry, rz], a, v)
    movel(p[x_c + 0.071964, y_c + -0.106095, z_c, rx, ry, rz], a, v)
    movel(p[x_c + 0.071955, y_c + -0.106092, z_c, rx, ry, rz], a, v)
    movel(p[x_c + 0.071948, y_c + -0.106090, z_c, rx, ry, rz], a, v)
    movel(p[x_c + 0.071945, y_c + -0.106090, z_c, rx, ry, rz], a, v)
    movel(p[x_c + 0.071943, y_c + -0.106093, z_c, rx, ry, rz], a, v)
    movel(p[x_c + 0.071945, y_c + -0.106098, z_c, rx, ry, rz], a, v)
    movel(p[x_c + 0.071949, y_c + -0.106104, z_c, rx, ry, rz], a, v)
    movel(p[x_c + 0.071955, y_c + -0.106113, z_c, rx, ry, rz], a, v)
    movel(p[x_c + 0.071965, y_c + -0.106125, z_c, rx, ry, rz], a, v)
    movel(p[x_c + 0.071977, y_c + -0.106138, z_c, rx, ry, rz], a, v)
    movel(p[x_c + 0.071991, y_c + -0.106153, z_c, rx, ry, rz], a, v)
    movel(p[x_c + 0.072008, y_c + -0.106171, z_c, rx, ry, rz], a, v)
    movel(p[x_c + 0.072028, y_c + -0.106191, z_c, rx, ry, rz], a, v)
    movel(p[x_c + 0.072051, y_c + -0.106214, z_c, rx, ry, rz], a, v)
    movel(p[x_c + 0.072076, y_c + -0.106238, z_c, rx, ry, rz], a, v)
    movel(p[x_c + 0.072104, y_c + -0.106265, z_c, rx, ry, rz], a, v)
    movel(p[x_c + 0.072135, y_c + -0.106294, z_c, rx, ry, rz], a, v)
    movel(p[x_c + 0.072168, y_c + -0.106325, z_c, rx, ry, rz], a, v)
    movel(p[x_c + 0.072204, y_c + -0.106359, z_c, rx, ry, rz], a, v)
    movel(p[x_c + 0.072243, y_c + -0.106395, z_c, rx, ry, rz], a, v)
